// TwinCAT 3 PLC project Testing
// ProgramVersion: 3.1.4026.26
// libraries:
//   Tc2_Standard, 3.4.7.0 (Beckhoff Automation GmbH)
//   Tc2_System, 3.10.2.0 (Beckhoff Automation GmbH)
//   [TcForge], 2.0.0.0 (Home)
//   TcUnit, 1.3.0.0 (www.tcunit.org)
//   [TcForgeExample], 2.0.0.0 (Home)
// project tree:
//   Testing/POUs/ FB_ControlLoopFixture.TcPOU, FB_AnalogOutputRestart_Probe.TcPOU, FB_AlarmRestart_Probe.TcPOU, FB_RpcContext_Probe.TcPOU, FB_OutputRestart_Probe.TcPOU, MAIN.TcPOU, FB_DeviceBase_Probe.TcPOU, FB_StateMachine_Probe.TcPOU
//   Testing/Tests/ FB_RegulatoryControl_Edge_Test.TcPOU, FB_RegulatoryControl_Test.TcPOU, FB_HysteresisControl_Test.TcPOU, FB_ExecutionContinuity_Test.TcPOU, FB_DigitalInputLifecycle_Test.TcPOU, FB_AlarmValidity_Test.TcPOU, FB_FilterLifecycle_Test.TcPOU, FB_PolicyNumeric_Test.TcPOU, FB_OutputConfiguration_Test.TcPOU, FB_IOQualityMonitor_Test.TcPOU, FB_InputLifecycle_Test.TcPOU, FB_OperatorMailbox_Test.TcPOU, FB_CommandValidation_Test.TcPOU, FB_ReferenceMachine_Test.TcPOU, FB_SequenceIntegrity_Test.TcPOU, FB_Foundation_Test.TcPOU, FB_CyclicFoundation_Test.TcPOU, FB_F_ValidateRequester_Test.TcPOU, FB_BitMatrix64_Test.TcPOU, FB_Permissives_Test.TcPOU, FB_Interlock_Test.TcPOU, FB_AlarmSimple_Test.TcPOU, FB_AlarmLimit_Test.TcPOU, FB_DeviceBase_Test.TcPOU, FB_LPF_FirstOrder_IIR_Test.TcPOU, FB_DigitalOutput_Test.TcPOU, FB_DigitalInput_Test.TcPOU, FB_TwoPosActuator_Test.TcPOU, FB_AnalogInput_Test.TcPOU, FB_AnalogOutput_Test.TcPOU, FB_AlarmThreshold_Test.TcPOU, FB_AlarmDeviation_Test.TcPOU, FB_Step_Test.TcPOU, FB_StateMachine_Test.TcPOU, FB_AssemblyStation_Test.TcPOU
//   Testing/ Testing.TcTTO
// (motion and I/O tree: see PLC project tcforge)
// real-time tasks:
//   TASK Testing: cycle T#10ms, priority 2, ADS port 351
//   TASK PlcTask: cycle T#10ms, priority 1, ADS port 350

CONFIGURATION Testing
    RESOURCE PLC ON TwinCAT3
        TASK Testing(INTERVAL := T#10ms, PRIORITY := 2);
        PROGRAM MAIN WITH Testing : MAIN;
    END_RESOURCE
END_CONFIGURATION

// ---- Testing/POUs/MAIN.TcPOU
PROGRAM MAIN
VAR
    controlLoopFixture : FB_ControlLoopFixture;
    regulatoryControlEdge : FB_RegulatoryControl_Edge_Test;
    regulatoryControl : FB_RegulatoryControl_Test;
    hysteresisControl : FB_HysteresisControl_Test;
    executionContinuity : FB_ExecutionContinuity_Test;
    digitalInputLifecycle : FB_DigitalInputLifecycle_Test;
    alarmValidity : FB_AlarmValidity_Test;
    filterLifecycle : FB_FilterLifecycle_Test;
    policyNumeric : FB_PolicyNumeric_Test;
    outputConfiguration : FB_OutputConfiguration_Test;
    ioQuality : FB_IOQualityMonitor_Test;
    inputLifecycle : FB_InputLifecycle_Test;
    simulation : FB_SimulationBridge;
    operatorMailbox : FB_OperatorMailbox_Test;
    rpcOutput : TcForge.FB_DigitalOutput;
    rpcUninitialized : TcForge.FB_DigitalOutput;
    enableRpcPump : BOOL := TRUE;
    commandValidation : FB_CommandValidation_Test;
    rpcContext : FB_RpcContext_Probe;
    assemblyStation : FB_AssemblyStation_Test;
    referenceMachine : FB_ReferenceMachine_Test;
    sequenceIntegrity : FB_SequenceIntegrity_Test;
    foundation : FB_Foundation_Test;
    cyclicFoundation : FB_CyclicFoundation_Test;
    fbValidateRequester_Test : FB_F_ValidateRequester_Test;
    fbBitMatrix64_Test       : FB_BitMatrix64_Test;
    fbPermissives_Test       : FB_Permissives_Test;
    fbInterlock_Test         : FB_Interlock_Test;
    fbAlarmSimple_Test       : FB_AlarmSimple_Test;
    fbAlarmLimit_Test        : FB_AlarmLimit_Test;
    fbDeviceBase_Test        : FB_DeviceBase_Test;
    fbLpfFirstOrder_Test     : FB_LPF_FirstOrder_IIR_Test;
    fbDigitalOutput_Test     : FB_DigitalOutput_Test;
    fbDigitalInput_Test      : FB_DigitalInput_Test;
    fbTwoPosActuator_Test    : FB_TwoPosActuator_Test;
    fbAnalogInput_Test       : FB_AnalogInput_Test;
    fbAnalogOutput_Test      : FB_AnalogOutput_Test;
    fbAlarmThreshold_Test    : FB_AlarmThreshold_Test;
    fbAlarmDeviation_Test    : FB_AlarmDeviation_Test;
    fbStep_Test              : FB_Step_Test;
    fbStateMachine_Test      : FB_StateMachine_Test;
END_VAR

controlLoopFixture();
simulation();
rpcContext();
IF enableRpcPump THEN rpcOutput(); END_IF;
TcUnit.RUN();

END_PROGRAM

// ---- Testing/POUs/FB_ControlLoopFixture.TcPOU
// Bench-only ADS surface for a generic first-order analog plant. There is no
// physical IO binding or operator command path. The Python runner writes the
// payload first and requestFrame last; the cyclic owner copies one complete
// frame, computes PID, publishes the result, then acknowledges appliedFrame.
FUNCTION_BLOCK FB_ControlLoopFixture
VAR
    // Test-writer fields. One monotonically increasing frame is accepted at a time.
    requestFrame    : UDINT;
    requestEnable   : BOOL;
    requestPv       : REAL;
    requestQuality  : USINT;
    requestSetpoint : REAL;

    // Stable until the next accepted frame or the 500 ms feed watchdog expires.
    appliedFrame    : UDINT;
    rejectedFrame   : UDINT;
    outputCv        : REAL;
    ready           : BOOL;
    reason          : TcForge.E_ControlReason;
    watchdogExpired : BOOL;
    watchdogTrips   : UDINT;
    ownerTask       : DINT;
    cycleCounter    : UDINT;

    _pid            : TcForge.FB_PID_Full;
    _cfg            : TcForge.ST_PID_Full_Cfg;
    _watchdog       : TON;
    _wasExpired     : BOOL;
    _activeEnable   : BOOL;
    _activePv       : REAL;
    _activeQuality  : TcForge.E_IO_Quality := TcForge.E_IO_Quality.UNKNOWN;
    _activeSp       : REAL;
    _frameFault     : BOOL;
    accepted        : BOOL;
    expectedFrame   : UDINT;
    pendingFrame    : UDINT;
END_VAR

ownerTask := Tc2_System.GETCURTASKINDEXEX();
cycleCounter := cycleCounter + 1;
accepted := FALSE;

// The final frame write is the commit marker. Old or skipped frame numbers
// invalidate the feed instead of leaving the previous regulator demand live.
IF appliedFrame = UDINT#16#FFFFFFFF THEN
    expectedFrame := 0;
ELSE
    expectedFrame := appliedFrame + 1;
END_IF;

IF requestFrame <> appliedFrame THEN
    IF requestFrame = expectedFrame THEN
        _activeEnable := requestEnable;
        _activePv := requestPv;
        _activeSp := requestSetpoint;
        _activeQuality := TcForge.E_IO_Quality.BAD;
        IF requestQuality = 2 THEN
            _activeQuality := TcForge.E_IO_Quality.GOOD;
        END_IF;

        pendingFrame := requestFrame;
        _frameFault := FALSE;
        accepted := TRUE;
    ELSE
        rejectedFrame := requestFrame;
        _frameFault := TRUE;
    END_IF;
END_IF;

_watchdog(IN := NOT accepted, PT := T#500MS);
watchdogExpired := _watchdog.Q;
IF watchdogExpired AND NOT _wasExpired THEN
    watchdogTrips := watchdogTrips + 1;
END_IF;
_wasExpired := watchdogExpired;

// Fixed, bounded tuning makes the test process generic and reproducible.
// The task period is read from the owning PLC task, not from ADS pacing.
_cfg.kp := 2.0;
_cfg.ki := 1.0;
_cfg.kd := 0.0;
_cfg.cvMin := 0.0;
_cfg.cvMax := 100.0;
_cfg.safeCv := 0.0;
_cfg.cycleTime := T#0MS;
_cfg.maxDt := T#100MS;

_pid(
    enable := _activeEnable AND NOT watchdogExpired AND NOT _frameFault,
    pv := _activePv,
    pvQuality := _activeQuality,
    setpoint := _activeSp,
    cfg := _cfg
);
outputCv := _pid.outCv;
ready := _pid.sts.ready;
reason := _pid.sts.reason;

// Publish acknowledgement after the CV and status for this frame.
IF accepted THEN
    appliedFrame := pendingFrame;
END_IF;

END_FUNCTION_BLOCK

// ---- Testing/Tests/FB_RegulatoryControl_Edge_Test.TcPOU
// Exercises mode transitions and boundary cases beyond the basic control suite.
FUNCTION_BLOCK FB_RegulatoryControl_Edge_Test EXTENDS TcUnit.FB_TestSuite
VAR
    _done : BOOL;
END_VAR

IF _done THEN
    RETURN;
END_IF;

StandardFormUsesIntegralTime();
DerivativeFiltersPvWithoutSetpointKick();
LowerLimitUnwindsOnReversal();
HoldAndTrackReleaseWithoutStep();
InvalidConfigurationAndTimingFailSafe();
TemperatureManualDutyAndPeriodEdit();
TemperatureRejectsInvalidConfiguration();
SwitchingPvRecoversAfterQualityLoss();
SwitchingContractClearsOldStatus();

_done := TRUE;

METHOD PRIVATE StandardFormUsesIntegralTime
VAR
    fb : TcForge.FB_PID_Full;
END_VAR
TEST('StandardFormUsesIntegralTime');

fb.cfg.standardForm := TRUE;
fb.cfg.kp := 2.0;
fb.cfg.integralTime := T#1S;
fb.cfg.cycleTime := T#100MS;
fb(enable := TRUE, pv := 0.0, pvQuality := TcForge.E_IO_Quality.GOOD, setpoint := 10.0);

AssertEquals_REAL(22.0, fb.outCv, 0.02, 'Standard form uses Kp/Ti for integral gain');
fb();
AssertEquals_REAL(24.0, fb.outCv, 0.02, 'Integral time advances the CV each cycle');

TEST_FINISHED();
END_METHOD

METHOD PRIVATE DerivativeFiltersPvWithoutSetpointKick
VAR
    fb : TcForge.FB_PID_Full;
END_VAR
TEST('DerivativeFiltersPvWithoutSetpointKick');

fb.cfg.kp := 0.0;
fb.cfg.kd := 1.0;
fb.cfg.derivativeTau := T#100MS;
fb.cfg.cvMin := -100.0;
fb.cfg.cycleTime := T#100MS;
fb(enable := TRUE, pv := 0.0, pvQuality := TcForge.E_IO_Quality.GOOD, setpoint := 0.0);

fb(pv := 1.0);
AssertEquals_REAL(-5.0, fb.outCv, 0.1, 'First-order filter halves the PV derivative');

fb(setpoint := 50.0);
AssertEquals_REAL(-2.5, fb.outCv, 0.1, 'Setpoint step does not enter PV derivative');

TEST_FINISHED();
END_METHOD

METHOD PRIVATE LowerLimitUnwindsOnReversal
VAR
    fb : TcForge.FB_PID_Full;
END_VAR
TEST('LowerLimitUnwindsOnReversal');

fb.cfg.kp := 0.0;
fb.cfg.ki := 1.0;
fb.cfg.cvMin := -2.0;
fb.cfg.cvMax := 2.0;
fb.cfg.cycleTime := T#100MS;
fb(enable := TRUE, pv := 0.0, pvQuality := TcForge.E_IO_Quality.GOOD, setpoint := -10.0);

fb();
fb();
AssertTrue(fb.sts.saturated, 'Further negative integration reports saturation');
AssertEquals_REAL(-2.0, fb.outCv, 0.02, 'Lower CV boundary is reached without windup');

fb(setpoint := 10.0);
AssertEquals_REAL(-1.0, fb.outCv, 0.02, 'Error reversal immediately unwinds integral');

TEST_FINISHED();
END_METHOD

METHOD PRIVATE HoldAndTrackReleaseWithoutStep
VAR
    fb : TcForge.FB_PID_Full;
END_VAR
TEST('HoldAndTrackReleaseWithoutStep');

fb.cfg.cycleTime := T#100MS;
fb(enable := TRUE, pv := 0.0, pvQuality := TcForge.E_IO_Quality.GOOD, setpoint := 20.0);
AssertEquals_REAL(20.0, fb.outCv, 0.01, 'Precondition: automatic CV');

fb(hold := TRUE, setpoint := 40.0);
AssertEquals_REAL(20.0, fb.outCv, 0.01, 'Hold keeps the last CV');
AssertTrue(fb.sts.reason = TcForge.E_ControlReason.Held, 'Hold mode is visible');

fb(track := TRUE, trackCv := 35.0);
AssertEquals_REAL(35.0, fb.outCv, 0.01, 'One-scan tracking takes the requested CV');

fb(track := FALSE, hold := FALSE);
AssertEquals_REAL(35.0, fb.outCv, 0.01, 'Automatic release uses tracked integral bias');

TEST_FINISHED();
END_METHOD

METHOD PRIVATE InvalidConfigurationAndTimingFailSafe
VAR
    fb : TcForge.FB_PID_Full;
END_VAR
TEST('InvalidConfigurationAndTimingFailSafe');

fb.cfg.cvMin := 100.0;
fb.cfg.cvMax := 0.0;
fb(enable := TRUE, pv := 0.0, pvQuality := TcForge.E_IO_Quality.GOOD, setpoint := 20.0);
AssertFalse(fb.sts.ready, 'Reversed CV limits cannot run');
AssertTrue(fb.sts.reason = TcForge.E_ControlReason.InvalidConfig, 'Invalid limits are diagnosed');
AssertEquals_REAL(0.0, fb.outCv, 0.001, 'Invalid configuration returns zero');

fb.cfg.cvMin := 0.0;
fb.cfg.cvMax := 100.0;
fb.cfg.cycleTime := T#2S;
fb();
AssertTrue(fb.sts.reason = TcForge.E_ControlReason.InvalidTiming, 'Oversize declared task interval is rejected');

fb.cfg.cycleTime := T#100MS;
fb();
AssertTrue(fb.sts.ready, 'Corrected timing starts a fresh controller');

fb(pvQuality := TcForge.E_IO_Quality.BAD);
AssertEquals_REAL(0.0, fb.outCv, 0.001, 'Bad quality immediately returns safe CV');

TEST_FINISHED();
END_METHOD

METHOD PRIVATE TemperatureManualDutyAndPeriodEdit
VAR
    fb : TcForge.FB_TempController;
    index : INT;
END_VAR
TEST('TemperatureManualDutyAndPeriodEdit');

fb.cfg.pid.cycleTime := T#100MS;
fb.cfg.pwmPeriod := T#1S;
fb(enable := TRUE, pv := 0.0, pvQuality := TcForge.E_IO_Quality.GOOD,
    setpoint := 25.0, manual := TRUE, manualDuty := 60.0);
AssertEquals_REAL(60.0, fb.outDuty, 0.01, 'Manual duty is applied as percent');

FOR index := 1 TO 7 DO
    fb();
END_FOR;
AssertFalse(fb.outOn, 'PWM reaches its OFF interval');

fb.cfg.pwmPeriod := T#2S;
fb();
AssertTrue(fb.outOn, 'Period edit restarts a bounded PWM window');

fb.cfg.pwmPeriod := T#50MS;
fb();
AssertFalse(fb.sts.ready, 'Too-short period is rejected');
AssertFalse(fb.outOn, 'Invalid period de-energizes PWM');

fb.cfg.pwmPeriod := T#1S;
fb();
AssertTrue(fb.sts.ready AND fb.outOn, 'Recovery starts a fresh ON window');

TEST_FINISHED();
END_METHOD

METHOD PRIVATE TemperatureRejectsInvalidConfiguration
VAR
    fb : TcForge.FB_TempController;
    invalid : REAL;
    bits : DWORD := DWORD#16#7F800001; // Signaling NaN; classify bits before comparison.
END_VAR
TEST('TemperatureRejectsInvalidConfiguration');

fb.cfg.pid.cvMin := -1.0;
fb.cfg.pid.cycleTime := T#100MS;
fb(enable := TRUE, pv := 0.0, pvQuality := TcForge.E_IO_Quality.GOOD, setpoint := 80.0);
AssertFalse(fb.sts.ready OR fb.outOn, 'Non-percent CV contract fails OFF');

fb.cfg.pid.cvMin := 0.0;
fb();
AssertTrue(fb.sts.ready AND fb.outOn, 'Valid percent contract can recover');

Tc2_System.MEMCPY(destAddr := ADR(invalid), srcAddr := ADR(bits), n := SIZEOF(invalid));
fb.cfg.standbySetpoint := invalid;
fb();
AssertFalse(fb.sts.ready OR fb.outOn, 'Nonfinite standby SP fails OFF even before use');

fb.cfg.standbySetpoint := 25.0;
fb();
AssertTrue(fb.sts.ready, 'Finite standby SP can recover');

TEST_FINISHED();
END_METHOD

METHOD PRIVATE SwitchingPvRecoversAfterQualityLoss
VAR
    fb : TcForge.FB_SwitchingPvPid;
END_VAR
TEST('SwitchingPvRecoversAfterQualityLoss');

fb.cfg.pv1.cycleTime := T#100MS;
fb.cfg.pv2.cycleTime := T#100MS;
fb(enable := TRUE, source := TcForge.E_PvSource.PV1,
    pv1 := 0.0, quality1 := TcForge.E_IO_Quality.GOOD, setpoint1 := 30.0,
    pv2 := 0.0, quality2 := TcForge.E_IO_Quality.BAD, setpoint2 := 40.0);
AssertEquals_REAL(30.0, fb.outCv, 0.01, 'PV1 is initially authoritative');

fb(source := TcForge.E_PvSource.PV2);
AssertFalse(fb.sts.ready, 'Selected bad PV cannot retain previous output');
AssertEquals_REAL(0.0, fb.outCv, 0.01, 'Bad selected PV returns common safe CV');

fb(quality2 := TcForge.E_IO_Quality.GOOD);
AssertEquals_REAL(40.0, fb.outCv, 0.01, 'Recovery uses fresh PV2 tuning, not stale CV');

TEST_FINISHED();
END_METHOD

METHOD PRIVATE SwitchingContractClearsOldStatus
VAR
    fb : TcForge.FB_SwitchingPvPid;
END_VAR
TEST('SwitchingContractClearsOldStatus');

fb.cfg.pv1.cycleTime := T#100MS;
fb.cfg.pv2.cycleTime := T#100MS;
fb(enable := TRUE, pv1 := 0.0, quality1 := TcForge.E_IO_Quality.GOOD, setpoint1 := 20.0);
AssertTrue(fb.sts.pid.ready, 'Precondition: PID status ready');

fb.cfg.pv2.cvMax := 80.0;
fb();
AssertFalse(fb.sts.ready OR fb.sts.pid.ready, 'Invalid shared contract clears old ready status');
AssertEquals_REAL(0.0, fb.outCv, 0.01, 'Invalid contract fails OFF');

fb.cfg.pv2.cvMax := 100.0;
fb();
AssertTrue(fb.sts.ready, 'Restored output contract can recover');

TEST_FINISHED();
END_METHOD

END_FUNCTION_BLOCK

// ---- Testing/Tests/FB_RegulatoryControl_Test.TcPOU
FUNCTION_BLOCK FB_RegulatoryControl_Test EXTENDS TcUnit.FB_TestSuite
VAR
    _done : BOOL;
END_VAR

IF _done THEN RETURN; END_IF;

BangBangMapsDemand();
PidProportionalAndReverse();
PidIntegralAndAntiWindup();
PidQualityAndManual();
PidSetpointAndCvRamps();
PidExceptionalInputFailsSafe();
TemperaturePwmAndStandby();
TemperatureQualityFailsOff();
SwitchingTracksCv();
SwitchingRejectsIncompatibleOutput();

_done := TRUE;

METHOD PRIVATE BangBangMapsDemand
VAR fb : TcForge.FB_BangBang; END_VAR
TEST('BangBangMapsDemand');
fb.cfg.hysteresis.low := 10.0;
fb.cfg.hysteresis.high := 20.0;
fb.cfg.lowValue := 5.0;
fb.cfg.highValue := 75.0;

fb(enable := TRUE, pv := 5.0, pvQuality := TcForge.E_IO_Quality.GOOD);
AssertTrue(fb.outDemand, 'Low PV requests the high mapped value');
AssertEquals_REAL(75.0, fb.outCv, 0.001, 'High value maps demand ON');

fb(pv := 20.0);
AssertFalse(fb.outDemand, 'High threshold clears demand');
AssertEquals_REAL(5.0, fb.outCv, 0.001, 'Low value maps demand OFF');

fb(pvQuality := TcForge.E_IO_Quality.BAD);
AssertFalse(fb.sts.ready, 'Bad quality invalidates mapped CV');
AssertEquals_REAL(0.0, fb.outCv, 0.001, 'Unusable mapping fails to zero');
TEST_FINISHED();
END_METHOD

METHOD PRIVATE PidProportionalAndReverse
VAR fb : TcForge.FB_PID_Full; END_VAR
TEST('PidProportionalAndReverse');
fb.cfg.kp := 2.0;
fb.cfg.cycleTime := T#100MS;
fb(enable := TRUE, pv := 20.0, pvQuality := TcForge.E_IO_Quality.GOOD, setpoint := 30.0);
AssertTrue(fb.sts.ready, 'Finite configured PID is ready');
AssertEquals_REAL(20.0, fb.outCv, 0.001, 'Direct P term drives CV');

fb.cfg.reverseActing := TRUE;
fb(pv := 30.0, setpoint := 20.0);
AssertFalse(fb.sts.ready, 'Tuning direction edit gets a safe scan');
fb();
AssertEquals_REAL(20.0, fb.outCv, 0.001, 'Reverse action changes error sign');
TEST_FINISHED();
END_METHOD

METHOD PRIVATE PidIntegralAndAntiWindup
VAR fb : TcForge.FB_PID_Full; END_VAR
TEST('PidIntegralAndAntiWindup');
fb.cfg.kp := 0.0;
fb.cfg.ki := 1.0;
fb.cfg.cycleTime := T#100MS;
fb(enable := TRUE, pv := 0.0, pvQuality := TcForge.E_IO_Quality.GOOD, setpoint := 10.0);
AssertEquals_REAL(1.0, fb.outCv, 0.001, 'Integral accumulates error times seconds');

fb();
AssertEquals_REAL(2.0, fb.outCv, 0.001, 'Integral advances by one output unit per scan');

fb.cfg.cvMax := 2.0;
fb();
AssertFalse(fb.sts.ready, 'CV limit edit invalidates old integral history');
fb();
AssertEquals_REAL(1.0, fb.outCv, 0.001, 'Reset history resumes from a fresh integral');
fb();
fb();
AssertTrue(fb.sts.saturated, 'Further integration is blocked at the CV limit');
AssertEquals_REAL(2.0, fb.outCv, 0.001, 'CV stays within the edited limit');
TEST_FINISHED();
END_METHOD

METHOD PRIVATE PidQualityAndManual
VAR fb : TcForge.FB_PID_Full; END_VAR
TEST('PidQualityAndManual');
fb.cfg.kp := 1.0;
fb.cfg.ki := 1.0;
fb.cfg.cycleTime := T#100MS;
fb(enable := TRUE, pv := 0.0, pvQuality := TcForge.E_IO_Quality.GOOD, setpoint := 10.0);
AssertTrue(fb.outCv > 0.0, 'Precondition: automatic CV is positive');

fb(manual := TRUE, manualCv := 40.0);
AssertEquals_REAL(40.0, fb.outCv, 0.001, 'Manual request is limited and published');
AssertTrue(fb.sts.reason = TcForge.E_ControlReason.Manual, 'Manual mode is visible');

fb(manual := FALSE);
AssertTrue(fb.outCv >= 40.0 AND fb.outCv < 42.0, 'Automatic resumes near tracked manual CV');

fb(pvQuality := TcForge.E_IO_Quality.BAD);
AssertEquals_REAL(0.0, fb.outCv, 0.001, 'Bad measurement immediately returns safe CV');
AssertFalse(fb.sts.ready, 'Bad quality cannot report ready');
TEST_FINISHED();
END_METHOD

METHOD PRIVATE PidSetpointAndCvRamps
VAR fb : TcForge.FB_PID_Full; END_VAR
TEST('PidSetpointAndCvRamps');
fb.cfg.kp := 1.0;
fb.cfg.spRateUp := 10.0;
fb.cfg.cvRateUp := 5.0;
fb.cfg.cycleTime := T#100MS;
fb(enable := TRUE, pv := 0.0, pvQuality := TcForge.E_IO_Quality.GOOD, setpoint := 0.0);

fb(setpoint := 10.0);
AssertEquals_REAL(1.0, fb.sts.spApplied, 0.001, 'SP ramp uses engineering units per second');
AssertEquals_REAL(0.5, fb.outCv, 0.001, 'CV ramp uses output units per second');
AssertTrue(fb.sts.spRamping AND fb.sts.cvRamping, 'Both active ramps are reported');
TEST_FINISHED();
END_METHOD

METHOD PRIVATE PidExceptionalInputFailsSafe
VAR
    fb : TcForge.FB_PID_Full;
    invalid : REAL;
    bits : DWORD := DWORD#16#7F800001; // Signaling NaN.
END_VAR
TEST('PidExceptionalInputFailsSafe');
fb.cfg.cycleTime := T#100MS;
fb(enable := TRUE, pv := 0.0, pvQuality := TcForge.E_IO_Quality.GOOD, setpoint := 20.0);
AssertTrue(fb.sts.ready, 'Precondition: valid PID');

Tc2_System.MEMCPY(destAddr := ADR(invalid), srcAddr := ADR(bits), n := SIZEOF(invalid));
fb(pv := invalid);
AssertFalse(fb.sts.ready, 'Signaling NaN is rejected before arithmetic');
AssertEquals_REAL(0.0, fb.outCv, 0.001, 'Rejected PV fails to safe CV');

fb(pv := 0.0);
AssertTrue(fb.sts.ready, 'Fresh finite PV can recover');
TEST_FINISHED();
END_METHOD

METHOD PRIVATE TemperaturePwmAndStandby
VAR fb : TcForge.FB_TempController; i : INT; END_VAR
TEST('TemperaturePwmAndStandby');
fb.cfg.pid.kp := 1.0;
fb.cfg.pid.cycleTime := T#100MS;
fb.cfg.pwmPeriod := T#1S;
fb.cfg.standbyEnabled := TRUE;
fb.cfg.standbySetpoint := 0.0;
fb(enable := TRUE, pv := 0.0, pvQuality := TcForge.E_IO_Quality.GOOD, setpoint := 50.0);
AssertEquals_REAL(50.0, fb.outDuty, 0.001, 'PID CV maps to 50 percent duty');
AssertTrue(fb.outOn, 'First half of PWM window is ON');

FOR i := 1 TO 5 DO fb(); END_FOR;
AssertFalse(fb.outOn, 'Second half of PWM window is OFF');

fb(standby := TRUE);
AssertTrue(fb.sts.standbyActive, 'Standby selects its own setpoint');
AssertEquals_REAL(0.0, fb.outDuty, 0.001, 'Standby zero setpoint removes heating demand');
AssertFalse(fb.outOn, 'Zero duty is OFF');
TEST_FINISHED();
END_METHOD

METHOD PRIVATE TemperatureQualityFailsOff
VAR fb : TcForge.FB_TempController; END_VAR
TEST('TemperatureQualityFailsOff');
fb.cfg.pid.cycleTime := T#100MS;
fb(enable := TRUE, pv := 0.0, pvQuality := TcForge.E_IO_Quality.GOOD, setpoint := 100.0);
AssertTrue(fb.outOn, 'Precondition: full-duty output ON');

fb(pvQuality := TcForge.E_IO_Quality.BAD);
AssertFalse(fb.outOn, 'Sensor loss removes PWM in the same scan');
AssertEquals_REAL(0.0, fb.outDuty, 0.001, 'Sensor loss returns zero duty');
AssertFalse(fb.sts.ready, 'Sensor loss cannot report ready');
TEST_FINISHED();
END_METHOD

METHOD PRIVATE SwitchingTracksCv
VAR fb : TcForge.FB_SwitchingPvPid; END_VAR
TEST('SwitchingTracksCv');
fb.cfg.pv1.cycleTime := T#100MS;
fb.cfg.pv2.cycleTime := T#100MS;
fb.cfg.pv2.ki := 1.0;
fb(enable := TRUE,
   source := TcForge.E_PvSource.PV1,
   pv1 := 0.0, quality1 := TcForge.E_IO_Quality.GOOD, setpoint1 := 20.0,
   pv2 := 0.0, quality2 := TcForge.E_IO_Quality.GOOD, setpoint2 := 40.0);
AssertEquals_REAL(20.0, fb.outCv, 0.001, 'PV1 regulates the shared output');

fb(source := TcForge.E_PvSource.PV2);
AssertTrue(fb.sts.sourceChanged, 'Selection change is published');
AssertEquals_REAL(20.0, fb.outCv, 0.001, 'PV2 tracks the previous CV for one scan');

fb();
AssertTrue(fb.outCv > 20.0 AND fb.outCv < 25.0, 'Selected PID resumes regulation');

fb(quality2 := TcForge.E_IO_Quality.BAD);
AssertFalse(fb.sts.ready, 'Selected bad PV invalidates the output');
AssertEquals_REAL(0.0, fb.outCv, 0.001, 'Selected bad PV uses the common safe CV');
TEST_FINISHED();
END_METHOD

METHOD PRIVATE SwitchingRejectsIncompatibleOutput
VAR fb : TcForge.FB_SwitchingPvPid; END_VAR
TEST('SwitchingRejectsIncompatibleOutput');
fb.cfg.pv1.cycleTime := T#100MS;
fb.cfg.pv2.cycleTime := T#100MS;
fb.cfg.pv2.cvMax := 80.0;
fb(enable := TRUE, pv1 := 0.0,
   quality1 := TcForge.E_IO_Quality.GOOD, setpoint1 := 50.0);
AssertFalse(fb.sts.ready, 'Different CV ranges cannot drive the same output');
AssertEquals_REAL(0.0, fb.outCv, 0.001, 'Mismatched output contract fails OFF');
TEST_FINISHED();
END_METHOD

END_FUNCTION_BLOCK

// ---- Testing/Tests/FB_HysteresisControl_Test.TcPOU
FUNCTION_BLOCK FB_HysteresisControl_Test EXTENDS TcUnit.FB_TestSuite
VAR
    _done : BOOL;
END_VAR

IF _done THEN
    RETURN;
END_IF;

DefaultRequiresConfiguration();
LowActingDeadband();
HighActingDeadband();
QualityLossClearsDemand();
ConfigChangeClearsDemand();
ExceptionalValuesFailOff();
DisableClearsDemand();

_done := TRUE;

METHOD PRIVATE DefaultRequiresConfiguration
VAR
    fb : TcForge.FB_HysteresisControl;
END_VAR
TEST('DefaultRequiresConfiguration');

fb(enable := TRUE, pv := 15.0, pvQuality := TcForge.E_IO_Quality.GOOD);
AssertFalse(fb.outDemand, 'Equal default thresholds cannot energize');
AssertTrue(fb.sts.reason = TcForge.E_HysteresisReason.InvalidConfig, 'Invalid defaults are visible');

fb.cfg.low := 10.0;
fb.cfg.high := 20.0;
fb();
AssertTrue(fb.sts.ready, 'Configured finite PV is ready');
AssertFalse(fb.outDemand, 'Startup inside the deadband starts OFF');

TEST_FINISHED();
END_METHOD

METHOD PRIVATE LowActingDeadband
VAR
    fb : TcForge.FB_HysteresisControl;
END_VAR
TEST('LowActingDeadband');

fb.cfg.low := 10.0;
fb.cfg.high := 20.0;
fb(enable := TRUE, pv := 5.0, pvQuality := TcForge.E_IO_Quality.GOOD);
AssertTrue(fb.outDemand, 'Heating demand turns ON below low threshold');

fb(pv := 15.0);
AssertTrue(fb.outDemand AND fb.sts.inDeadband, 'Demand holds ON inside deadband');

fb(pv := 20.0);
AssertFalse(fb.outDemand, 'Demand turns OFF at high threshold');

fb(pv := 15.0);
AssertFalse(fb.outDemand, 'Deadband also retains OFF state');

fb(pv := 10.0);
AssertTrue(fb.outDemand, 'Demand turns ON at low threshold');

TEST_FINISHED();
END_METHOD

METHOD PRIVATE HighActingDeadband
VAR
    fb : TcForge.FB_HysteresisControl;
END_VAR
TEST('HighActingDeadband');

fb.cfg.low := 10.0;
fb.cfg.high := 20.0;
fb.cfg.onBelowLow := FALSE;
fb(enable := TRUE, pv := 25.0, pvQuality := TcForge.E_IO_Quality.GOOD);
AssertTrue(fb.outDemand, 'Cooling demand turns ON above high threshold');

fb(pv := 15.0);
AssertTrue(fb.outDemand, 'Cooling demand holds ON inside deadband');

fb(pv := 10.0);
AssertFalse(fb.outDemand, 'Cooling demand turns OFF at low threshold');

fb(pv := 15.0);
AssertFalse(fb.outDemand, 'Cooling deadband retains OFF state');

TEST_FINISHED();
END_METHOD

METHOD PRIVATE QualityLossClearsDemand
VAR
    fb : TcForge.FB_HysteresisControl;
END_VAR
TEST('QualityLossClearsDemand');

fb.cfg.low := 10.0;
fb.cfg.high := 20.0;
fb(enable := TRUE, pv := 5.0, pvQuality := TcForge.E_IO_Quality.GOOD);
AssertTrue(fb.outDemand, 'Precondition: demand ON');

fb(pvQuality := TcForge.E_IO_Quality.BAD);
AssertFalse(fb.outDemand, 'Quality loss removes demand in the same scan');
AssertTrue(fb.sts.reason = TcForge.E_HysteresisReason.BadQuality, 'Quality loss is diagnosed');

fb(pv := 15.0, pvQuality := TcForge.E_IO_Quality.GOOD);
AssertFalse(fb.outDemand, 'Recovery inside deadband cannot restore stale ON intent');

fb(pv := 10.0);
AssertTrue(fb.outDemand, 'Fresh threshold crossing may demand ON');

TEST_FINISHED();
END_METHOD

METHOD PRIVATE ConfigChangeClearsDemand
VAR
    fb : TcForge.FB_HysteresisControl;
END_VAR
TEST('ConfigChangeClearsDemand');

fb.cfg.low := 10.0;
fb.cfg.high := 20.0;
fb(enable := TRUE, pv := 5.0, pvQuality := TcForge.E_IO_Quality.GOOD);
AssertTrue(fb.outDemand, 'Precondition: old recipe demands ON');

fb.cfg.low := 0.0;
fb(pv := 5.0);
AssertFalse(fb.outDemand, 'Changed threshold cannot inherit old ON state in deadband');

fb.cfg.onBelowLow := FALSE;
fb();
AssertFalse(fb.outDemand, 'Changed direction also starts from OFF');

fb(pv := 20.0);
AssertTrue(fb.outDemand, 'New direction can turn ON at its threshold');

TEST_FINISHED();
END_METHOD

METHOD PRIVATE ExceptionalValuesFailOff
VAR
    fb : TcForge.FB_HysteresisControl;
    invalid : REAL;
    bits : DWORD := DWORD#16#7F800001; // Signaling NaN; never compare as REAL.
END_VAR
TEST('ExceptionalValuesFailOff');

fb.cfg.low := 10.0;
fb.cfg.high := 20.0;
fb(enable := TRUE, pv := 5.0, pvQuality := TcForge.E_IO_Quality.GOOD);
AssertTrue(fb.outDemand, 'Precondition: demand ON');

Tc2_System.MEMCPY(destAddr := ADR(invalid), srcAddr := ADR(bits), n := SIZEOF(invalid));
fb(pv := invalid);
AssertFalse(fb.outDemand, 'Nonfinite PV fails OFF without a floating-point comparison');
AssertTrue(fb.sts.reason = TcForge.E_HysteresisReason.InvalidValue, 'Nonfinite PV is diagnosed');

fb(pv := 5.0);
AssertTrue(fb.outDemand, 'Fresh valid PV at threshold may restore demand');

fb.cfg.low := invalid;
fb();
AssertFalse(fb.outDemand, 'Nonfinite threshold fails OFF');
AssertTrue(fb.sts.reason = TcForge.E_HysteresisReason.InvalidConfig, 'Bad threshold is diagnosed');

TEST_FINISHED();
END_METHOD

METHOD PRIVATE DisableClearsDemand
VAR
    fb : TcForge.FB_HysteresisControl;
END_VAR
TEST('DisableClearsDemand');

fb.cfg.low := 10.0;
fb.cfg.high := 20.0;
fb(enable := TRUE, pv := 5.0, pvQuality := TcForge.E_IO_Quality.GOOD);
AssertTrue(fb.outDemand, 'Precondition: demand ON');

fb(enable := FALSE);
AssertFalse(fb.outDemand, 'Disable removes demand');
AssertTrue(fb.sts.reason = TcForge.E_HysteresisReason.Disabled, 'Disabled status is explicit');

fb(enable := TRUE, pv := 15.0);
AssertFalse(fb.outDemand, 'Re-enable inside deadband remains OFF');

TEST_FINISHED();
END_METHOD

END_FUNCTION_BLOCK

// ---- Testing/Tests/FB_ExecutionContinuity_Test.TcPOU
FUNCTION_BLOCK FB_ExecutionContinuity_Test EXTENDS TcUnit.FB_TestSuite
VAR done : BOOL; END_VAR

IF NOT done THEN
InitialObservationEstablishesBaseline();
ContinuousAndRepeatedCycle();
SkippedScanRequiresRecovery();
OnlineChangeDetectedWithoutGap();
TaskChangeAndInvalidContext();
CounterWrapAndReset();
CompatibleChangePreservesExecution();
CompatibleChangeCannotMaskGap();
CompatiblePolicyCannotMaskOwnerFailure();
done := TRUE; END_IF;

METHOD InitialObservationEstablishesBaseline
VAR fb : TcForge.FB_ExecutionContinuity; END_VAR
TEST('InitialObservationEstablishesBaseline');
fb(taskIndex := 1, cycleCounter := 99, onlineChangeCounter := 3); AssertFalse(Condition := fb.interrupted, Message := 'First sample establishes baseline');
TEST_FINISHED();
END_METHOD

METHOD ContinuousAndRepeatedCycle
VAR fb : TcForge.FB_ExecutionContinuity; END_VAR
TEST('ContinuousAndRepeatedCycle');
fb(taskIndex := 1, cycleCounter := 99); fb(cycleCounter := 100); AssertFalse(Condition := fb.interrupted, Message := 'Next scan continues'); fb(); AssertFalse(Condition := fb.interrupted, Message := 'Same scan observation is idempotent');
TEST_FINISHED();
END_METHOD

METHOD SkippedScanRequiresRecovery
VAR fb : TcForge.FB_ExecutionContinuity; END_VAR
TEST('SkippedScanRequiresRecovery');
fb(taskIndex := 1, cycleCounter := 99); fb(cycleCounter := 101); AssertTrue(Condition := fb.interrupted, Message := 'Missed execution detected'); fb(cycleCounter := 102); AssertFalse(Condition := fb.interrupted, Message := 'Caller must latch recovery; event is one scan');
TEST_FINISHED();
END_METHOD

METHOD OnlineChangeDetectedWithoutGap
VAR fb : TcForge.FB_ExecutionContinuity; END_VAR
TEST('OnlineChangeDetectedWithoutGap');
fb(taskIndex := 1, cycleCounter := 99, onlineChangeCounter := 3); fb(cycleCounter := 100, onlineChangeCounter := 4); AssertTrue(Condition := fb.interrupted, Message := 'Implementation-only online change detected');
TEST_FINISHED();
END_METHOD

METHOD TaskChangeAndInvalidContext
VAR fb : TcForge.FB_ExecutionContinuity; END_VAR
TEST('TaskChangeAndInvalidContext');
fb(taskIndex := 1, cycleCounter := 99); fb(taskIndex := 2, cycleCounter := 100); AssertTrue(Condition := fb.interrupted, Message := 'Different owner detected'); fb(taskIndex := 0); AssertTrue(Condition := fb.interrupted, Message := 'RPC or invalid context rejected');
TEST_FINISHED();
END_METHOD

METHOD CounterWrapAndReset
VAR fb : TcForge.FB_ExecutionContinuity; END_VAR
TEST('CounterWrapAndReset');
fb(taskIndex := 1, cycleCounter := UDINT#16#FFFFFFFF); fb(cycleCounter := 0); AssertFalse(Condition := fb.interrupted, Message := 'Natural wrap is continuous'); fb(cycleCounter := 99); fb(cycleCounter := 0); AssertTrue(Condition := fb.interrupted, Message := 'Counter discontinuity detected');
TEST_FINISHED();
END_METHOD

METHOD CompatibleChangePreservesExecution
VAR fb : TcForge.FB_ExecutionContinuity; END_VAR
TEST('CompatibleChangePreservesExecution');
fb(taskIndex := 1, cycleCounter := 99, onlineChangeCounter := 3, recoverOnOnlineChange := FALSE);
fb(cycleCounter := 100, onlineChangeCounter := 4);
AssertTrue(Condition := fb.onlineChanged, Message := 'Change remains observable');
AssertFalse(Condition := fb.executionInterrupted, Message := 'Online edit is not an execution gap');
AssertFalse(Condition := fb.interrupted, Message := 'Explicit compatible-edit policy preserves execution');
fb(cycleCounter := 101);
AssertFalse(Condition := fb.onlineChanged, Message := 'Change notification is a pulse');
TEST_FINISHED();
END_METHOD

METHOD CompatibleChangeCannotMaskGap
VAR fb : TcForge.FB_ExecutionContinuity; END_VAR
TEST('CompatibleChangeCannotMaskGap');
fb(taskIndex := 1, cycleCounter := 99, onlineChangeCounter := 3, recoverOnOnlineChange := FALSE);
fb(cycleCounter := 101, onlineChangeCounter := 4);
AssertTrue(Condition := fb.onlineChanged, Message := 'Simultaneous online edit observed');
AssertTrue(Condition := fb.executionInterrupted, Message := 'Gap remains a gap during online edit');
AssertTrue(Condition := fb.interrupted, Message := 'Compatible-edit policy cannot suppress recovery');
TEST_FINISHED();
END_METHOD

METHOD CompatiblePolicyCannotMaskOwnerFailure
VAR fb : TcForge.FB_ExecutionContinuity; END_VAR
TEST('CompatiblePolicyCannotMaskOwnerFailure');
fb(taskIndex := 1, cycleCounter := 99, recoverOnOnlineChange := FALSE);
fb(taskIndex := 2, cycleCounter := 100);
AssertTrue(Condition := fb.interrupted, Message := 'Owner conflict still requires recovery');
fb(taskIndex := 0);
AssertTrue(Condition := fb.executionInterrupted, Message := 'Invalid context still fails closed');
TEST_FINISHED();
END_METHOD

END_FUNCTION_BLOCK

// ---- Testing/Tests/FB_DigitalInputLifecycle_Test.TcPOU
FUNCTION_BLOCK FB_DigitalInputLifecycle_Test EXTENDS TcUnit.FB_TestSuite
VAR
BadQualityCannotCompleteRising_fb : TcForge.FB_DigitalInput;
BadQualityCannotCompleteRising_clock : TON;
BadQualityCannotCompleteRising_phase : UINT;
BadQualityCannotCompleteRising_done : BOOL;
BadQualityCannotCompleteFalling_fb : TcForge.FB_DigitalInput;
BadQualityCannotCompleteFalling_clock : TON;
BadQualityCannotCompleteFalling_phase : UINT;
BadQualityCannotCompleteFalling_done : BOOL;
ConfigChangeDiscardsDebounceCredit_fb : TcForge.FB_DigitalInput;
ConfigChangeDiscardsDebounceCredit_clock : TON;
ConfigChangeDiscardsDebounceCredit_phase : UINT;
ConfigChangeDiscardsDebounceCredit_done : BOOL;
_instantDone : BOOL;
END_VAR


BadQualityCannotCompleteRising();
BadQualityCannotCompleteFalling();
ConfigChangeDiscardsDebounceCredit();
IF NOT _instantDone THEN ReassignmentAndInvalidConfigHold(); _instantDone := TRUE; END_IF;

METHOD BadQualityCannotCompleteRising
IF BadQualityCannotCompleteRising_done THEN RETURN; END_IF;
TEST('BadQualityCannotCompleteRising');
CASE BadQualityCannotCompleteRising_phase OF
0:
    BadQualityCannotCompleteRising_fb(inSignal := FALSE);
    BadQualityCannotCompleteRising_fb.cfg.debounceOn := T#80MS; BadQualityCannotCompleteRising_fb.cfg.debounceOff := T#80MS;
    BadQualityCannotCompleteRising_fb(inSignal := TRUE);
    BadQualityCannotCompleteRising_fb(inpQuality := TcForge.E_IO_Quality.BAD);
    BadQualityCannotCompleteRising_phase := 1;
1:
    BadQualityCannotCompleteRising_clock(IN := TRUE, PT := T#150MS); BadQualityCannotCompleteRising_fb();
    IF BadQualityCannotCompleteRising_clock.Q THEN
        AssertEquals_BOOL(Expected := FALSE, Actual := BadQualityCannotCompleteRising_fb.sts.value, Message := 'Invalid elapsed time must hold established state');
        AssertFalse(Condition := BadQualityCannotCompleteRising_fb.sts.risingEdge OR BadQualityCannotCompleteRising_fb.sts.fallingEdge, Message := 'Invalid sample cannot emit edges');
        BadQualityCannotCompleteRising_clock(IN := FALSE); BadQualityCannotCompleteRising_fb(inpQuality := TcForge.E_IO_Quality.GOOD);
        AssertEquals_BOOL(Expected := FALSE, Actual := BadQualityCannotCompleteRising_fb.sts.value, Message := 'Recovery starts a full fresh transition delay');
        BadQualityCannotCompleteRising_phase := 2;
    END_IF;
2:
    BadQualityCannotCompleteRising_clock(IN := TRUE, PT := T#30MS); BadQualityCannotCompleteRising_fb();
    IF BadQualityCannotCompleteRising_clock.Q THEN
        AssertEquals_BOOL(Expected := FALSE, Actual := BadQualityCannotCompleteRising_fb.sts.value, Message := 'Partial fresh delay cannot complete transition');
        BadQualityCannotCompleteRising_clock(IN := FALSE); BadQualityCannotCompleteRising_phase := 3;
    END_IF;
3:
    BadQualityCannotCompleteRising_clock(IN := TRUE, PT := T#150MS); BadQualityCannotCompleteRising_fb();
    IF BadQualityCannotCompleteRising_clock.Q THEN
        AssertEquals_BOOL(Expected := TRUE, Actual := BadQualityCannotCompleteRising_fb.sts.value, Message := 'Full fresh delay completes transition');
        BadQualityCannotCompleteRising_done := TRUE; TEST_FINISHED();
    END_IF;
END_CASE;
END_METHOD

METHOD BadQualityCannotCompleteFalling
IF BadQualityCannotCompleteFalling_done THEN RETURN; END_IF;
TEST('BadQualityCannotCompleteFalling');
CASE BadQualityCannotCompleteFalling_phase OF
0:
    BadQualityCannotCompleteFalling_fb(inSignal := TRUE);
    BadQualityCannotCompleteFalling_fb.cfg.debounceOn := T#80MS; BadQualityCannotCompleteFalling_fb.cfg.debounceOff := T#80MS;
    BadQualityCannotCompleteFalling_fb(inSignal := FALSE);
    BadQualityCannotCompleteFalling_fb(inpQuality := TcForge.E_IO_Quality.BAD);
    BadQualityCannotCompleteFalling_phase := 1;
1:
    BadQualityCannotCompleteFalling_clock(IN := TRUE, PT := T#150MS); BadQualityCannotCompleteFalling_fb();
    IF BadQualityCannotCompleteFalling_clock.Q THEN
        AssertEquals_BOOL(Expected := TRUE, Actual := BadQualityCannotCompleteFalling_fb.sts.value, Message := 'Invalid elapsed time must hold established state');
        AssertFalse(Condition := BadQualityCannotCompleteFalling_fb.sts.risingEdge OR BadQualityCannotCompleteFalling_fb.sts.fallingEdge, Message := 'Invalid sample cannot emit edges');
        BadQualityCannotCompleteFalling_clock(IN := FALSE); BadQualityCannotCompleteFalling_fb(inpQuality := TcForge.E_IO_Quality.GOOD);
        AssertEquals_BOOL(Expected := TRUE, Actual := BadQualityCannotCompleteFalling_fb.sts.value, Message := 'Recovery starts a full fresh transition delay');
        BadQualityCannotCompleteFalling_phase := 2;
    END_IF;
2:
    BadQualityCannotCompleteFalling_clock(IN := TRUE, PT := T#30MS); BadQualityCannotCompleteFalling_fb();
    IF BadQualityCannotCompleteFalling_clock.Q THEN
        AssertEquals_BOOL(Expected := TRUE, Actual := BadQualityCannotCompleteFalling_fb.sts.value, Message := 'Partial fresh delay cannot complete transition');
        BadQualityCannotCompleteFalling_clock(IN := FALSE); BadQualityCannotCompleteFalling_phase := 3;
    END_IF;
3:
    BadQualityCannotCompleteFalling_clock(IN := TRUE, PT := T#150MS); BadQualityCannotCompleteFalling_fb();
    IF BadQualityCannotCompleteFalling_clock.Q THEN
        AssertEquals_BOOL(Expected := FALSE, Actual := BadQualityCannotCompleteFalling_fb.sts.value, Message := 'Full fresh delay completes transition');
        BadQualityCannotCompleteFalling_done := TRUE; TEST_FINISHED();
    END_IF;
END_CASE;
END_METHOD

METHOD ConfigChangeDiscardsDebounceCredit
IF ConfigChangeDiscardsDebounceCredit_done THEN RETURN; END_IF;
TEST('ConfigChangeDiscardsDebounceCredit');
CASE ConfigChangeDiscardsDebounceCredit_phase OF
0:
    ConfigChangeDiscardsDebounceCredit_fb.cfg.debounceOn := T#100MS;
    ConfigChangeDiscardsDebounceCredit_fb(inSignal := TRUE);
    ConfigChangeDiscardsDebounceCredit_phase := 1;
1:
    ConfigChangeDiscardsDebounceCredit_clock(IN := TRUE, PT := T#60MS); ConfigChangeDiscardsDebounceCredit_fb();
    IF ConfigChangeDiscardsDebounceCredit_clock.Q THEN
        ConfigChangeDiscardsDebounceCredit_fb.cfg.debounceOn := T#80MS;
        ConfigChangeDiscardsDebounceCredit_fb(); ConfigChangeDiscardsDebounceCredit_clock(IN := FALSE);
        ConfigChangeDiscardsDebounceCredit_phase := 2;
    END_IF;
2:
    ConfigChangeDiscardsDebounceCredit_clock(IN := TRUE, PT := T#30MS); ConfigChangeDiscardsDebounceCredit_fb();
    IF ConfigChangeDiscardsDebounceCredit_clock.Q THEN
        AssertFalse(Condition := ConfigChangeDiscardsDebounceCredit_fb.sts.value, Message := 'New delay cannot inherit old timer credit');
        ConfigChangeDiscardsDebounceCredit_done := TRUE; TEST_FINISHED();
    END_IF;
END_CASE;
END_METHOD

METHOD ReassignmentAndInvalidConfigHold
VAR fb : TcForge.FB_DigitalInput; END_VAR

TEST('ReassignmentAndInvalidConfigHold');
fb(inSignal := TRUE); AssertTrue(Condition := fb.sts.value, Message := 'Fixture has established TRUE');
fb(inpQuality := TcForge.E_IO_Quality.UNKNOWN); fb.cfg.invert := TRUE; fb();
AssertTrue(Condition := fb.sts.value, Message := 'Inversion cannot reinterpret invalid held raw');
AssertFalse(Condition := fb.sts.risingEdge OR fb.sts.fallingEdge, Message := 'Config edit under bad quality has no edge');
fb.ReassignInput();
AssertEquals_INT(Expected := 0, Actual := fb.sts.quality, Message := 'Reassignment immediately invalidates old source');
AssertFalse(Condition := fb.sts.value OR fb.sts.rawValue OR fb.sts.risingEdge OR fb.sts.fallingEdge, Message := 'Reassignment clears old history without an edge');
fb(); AssertEquals_INT(Expected := 0, Actual := fb.sts.quality, Message := 'Unknown adapter quality remains unknown');
fb(inpQuality := TcForge.E_IO_Quality.GOOD, inSignal := FALSE);
AssertTrue(Condition := fb.sts.value AND fb.sts.risingEdge, Message := 'Fresh source is conditioned using current inversion');
TEST_FINISHED();
END_METHOD

END_FUNCTION_BLOCK

// ---- Testing/Tests/FB_AlarmValidity_Test.TcPOU
FUNCTION_BLOCK FB_AlarmValidity_Test EXTENDS TcUnit.FB_TestSuite
VAR
    done : BOOL;
    restoredUnacked : FB_AlarmRestart_Probe;
    restoredAcked : FB_AlarmRestart_Probe;
    criteriaThreshold : TcForge.FB_AlarmThreshold;
    criteriaDeviation : TcForge.FB_AlarmDeviation;
    criteriaPhase : UINT;
    beforeChange : TON;
    afterChange : TON;
    reassignedRate : TcForge.FB_AlarmRateOfChange;
    severityAlarm : TcForge.FB_AlarmSimple;
    signalingAlarm : TcForge.FB_AlarmThreshold;
    recovery : TcForge.FB_AlarmSimple;
    phase : UINT;
    waitTimer : TON;
    clearTimer : TON;
    device0 : TcForge.FB_AlarmThreshold;
    device1 : TcForge.FB_AlarmThreshold;
    device2 : TcForge.FB_AlarmSimple;
    device3 : TcForge.FB_AlarmSimple;
    device4 : TcForge.FB_AlarmDeviation;
    device5 : TcForge.FB_AlarmDeviation;
    device6 : TcForge.FB_AlarmRateOfChange;
    device7 : TcForge.FB_AlarmRateOfChange;
    device8 : TcForge.FB_AlarmRateOfChange;
    device9 : TcForge.FB_AlarmLimit;
END_VAR

IF NOT done THEN
InvalidInputPreservesAlarm();
RestoredLatchPublishesSeverity();
RestoredAcknowledgmentNeedsClearEvidence();
InvalidConfigPreservesLatch();
RequireAckChangePreservesLatch();
SimpleValidityGate();
DeviationExtremeArithmetic();
DeviationRejectsBadBounds();
RateExtremeArithmetic();
RateRecoveryNeedsTwoSamples();
RateConfigReseedsHistory();
LimitRollupValidity();
InvalidSeverityPreservesAlarm();
SignalingNaNIsClassified();
RateReassignmentDropsHistory();
done := TRUE;
END_IF;
RecoveryHonorsFreshClearDelay();
CriteriaChangeRestartsTripDelay();

METHOD PRIVATE RestoredLatchPublishesSeverity
TEST('RestoredLatchPublishesSeverity');
restoredUnacked.SeedSavedLatch(acknowledged := FALSE);
restoredUnacked.cfg.common.bEnable := TRUE;
restoredUnacked.cfg.common.bRequireAck := TRUE;
restoredUnacked.cfg.common.eSeverity := TcForge.E_AlarmSeverity.SHUTDOWN;
restoredUnacked(inpActive := FALSE, inpValid := FALSE);
AssertTrue(restoredUnacked.sts.active AND restoredUnacked.sts.latched, 'Restored unacked latch remains active without valid input');
AssertFalse(restoredUnacked.sts.valid, 'Restored latch is not valid process evidence');
AssertEquals_DINT(TcForge.E_AlarmSeverity.SHUTDOWN, restoredUnacked.sts.eSeverity, 'Startup publishes configured severity despite invalid input');
restoredUnacked.cfg.common.eSeverity := TcForge.E_AlarmSeverity.INFO;
restoredUnacked();
AssertEquals_DINT(TcForge.E_AlarmSeverity.SHUTDOWN, restoredUnacked.sts.eSeverity, 'Later invalid evaluation preserves established severity');
restoredUnacked(inpValid := TRUE);
AssertTrue(restoredUnacked.sts.active AND restoredUnacked.sts.latched, 'Valid clear evidence alone cannot erase an unacked restored latch');
restoredUnacked.Ack(); restoredUnacked();
AssertFalse(restoredUnacked.sts.active, 'Explicit Ack and valid clear release restored latch');
TEST_FINISHED();
END_METHOD

METHOD PRIVATE RestoredAcknowledgmentNeedsClearEvidence
TEST('RestoredAcknowledgmentNeedsClearEvidence');
restoredAcked.SeedSavedLatch(acknowledged := TRUE);
restoredAcked.cfg.common.bEnable := TRUE;
restoredAcked.cfg.common.bRequireAck := TRUE;
restoredAcked.cfg.common.eSeverity := TcForge.E_AlarmSeverity.CRITICAL;
restoredAcked(inpActive := FALSE, inpValid := FALSE);
AssertTrue(restoredAcked.sts.active AND restoredAcked.sts.acked, 'Restored acknowledgment cannot clear alarm with invalid evidence');
AssertFalse(restoredAcked.sts.latched, 'Restored acknowledged alarm does not demand another Ack');
AssertEquals_DINT(TcForge.E_AlarmSeverity.CRITICAL, restoredAcked.sts.eSeverity, 'Acknowledged restored alarm retains meaningful startup severity');
restoredAcked(inpValid := TRUE);
AssertFalse(restoredAcked.sts.active OR restoredAcked.sts.acked, 'Valid clear evidence releases restored acknowledged latch without a second Ack');
TEST_FINISHED();
END_METHOD

METHOD PRIVATE InvalidInputPreservesAlarm
VAR bits : TcForge.U_IoRaw_Out; tripped, cleared : LTIME; END_VAR
TEST('InvalidInputPreservesAlarm');
device0.cfg.common.bEnable := TRUE; device0.cfg.bFailHigh := TRUE;
device0.cfg.common.eSeverity := TcForge.E_AlarmSeverity.CRITICAL;
device0(inpValue := 10.0); tripped := device0.sts.tsTripped; cleared := device0.sts.tsCleared;
bits.dw := DWORD#16#7FC00000; device0(inpValue := bits.fReal);
AssertTrue(device0.sts.active, 'NaN cannot clear active alarm');
AssertFalse(device0.sts.valid, 'NaN evaluation is invalid');
AssertEquals_DINT(TcForge.E_AlarmEvaluation.InvalidInput, device0.sts.evaluationState, 'NaN classified without FPU operation');
AssertEquals_DINT(TcForge.E_AlarmSeverity.CRITICAL, device0.sts.eSeverity, 'Established severity preserved');
AssertTrue(device0.sts.tsTripped = tripped AND device0.sts.tsCleared = cleared, 'Invalid evaluation creates no alarm edges');
TEST_FINISHED();
END_METHOD

METHOD PRIVATE InvalidConfigPreservesLatch
VAR bits : TcForge.U_IoRaw_Out; tripped, cleared : LTIME; END_VAR
TEST('InvalidConfigPreservesLatch');
device1.cfg.common.bEnable := TRUE; device1.cfg.bFailHigh := TRUE; device1.cfg.common.bRequireAck := TRUE;
device1(inpValue := 10.0);
bits.dw := DWORD#16#7FC00000; device1.cfg.fThreshold := bits.fReal;
device1(); device1.Ack(); device1();
AssertTrue(device1.sts.active, 'Ack during invalid config cannot clear latch');
AssertTrue(device1.sts.acked, 'Ack is recorded while evaluation is invalid');
device1.cfg.fThreshold := 20.0; device1();
AssertFalse(device1.sts.active, 'Valid clear evidence releases acknowledged latch');
TEST_FINISHED();
END_METHOD

METHOD PRIVATE RequireAckChangePreservesLatch
VAR bits : TcForge.U_IoRaw_Out; tripped, cleared : LTIME; END_VAR
TEST('RequireAckChangePreservesLatch');
device2.cfg.common.bEnable := TRUE; device2.cfg.common.bRequireAck := TRUE;
device2(inpActive := TRUE); device2.cfg.common.bRequireAck := FALSE; device2(inpActive := FALSE);
AssertTrue(device2.sts.active AND device2.sts.latched, 'Changing future latch policy does not erase unacked trip');
device2.Ack(); device2(); AssertFalse(device2.sts.active, 'Ack and valid clear release old latch');
TEST_FINISHED();
END_METHOD

METHOD PRIVATE SimpleValidityGate
VAR bits : TcForge.U_IoRaw_Out; tripped, cleared : LTIME; END_VAR
TEST('SimpleValidityGate');
device3.cfg.common.bEnable := TRUE; device3(inpActive := TRUE);
device3(inpActive := FALSE, inpValid := FALSE);
AssertTrue(device3.sts.active, 'Missing digital quality holds established alarm');
AssertFalse(device3.sts.valid, 'Missing quality is visible');
device3(inpValid := TRUE); AssertFalse(device3.sts.active, 'Valid clear evidence releases nonlatched alarm');
TEST_FINISHED();
END_METHOD

METHOD PRIVATE DeviationExtremeArithmetic
VAR bits : TcForge.U_IoRaw_Out; tripped, cleared : LTIME; END_VAR
TEST('DeviationExtremeArithmetic');
device4.cfg.common.bEnable := TRUE; device4.cfg.bUseSetpoint := TRUE;
device4.cfg.fHighLimit := 3.0E38; device4.cfg.fLowLimit := 3.0E38;
device4(inpPv := 3.0E38, inpSetpoint := 3.0E38);
AssertTrue(device4.sts.valid, 'Finite extremes use wide intermediate bounds');
AssertFalse(device4.sts.active, 'Large valid setpoint window contains PV');
TEST_FINISHED();
END_METHOD

METHOD PRIVATE DeviationRejectsBadBounds
VAR bits : TcForge.U_IoRaw_Out; tripped, cleared : LTIME; END_VAR
TEST('DeviationRejectsBadBounds');
device5.cfg.common.bEnable := TRUE; device5.cfg.fHighLimit := 1.0; device5.cfg.fLowLimit := 2.0; device5();
AssertEquals_DINT(TcForge.E_AlarmEvaluation.InvalidConfig, device5.sts.evaluationState, 'Reversed absolute bounds rejected');
device5.cfg.bUseSetpoint := TRUE; device5.cfg.fLowLimit := -1.0; device5();
AssertFalse(device5.sts.valid, 'Negative setpoint deviation rejected');
device5.cfg.fLowLimit := 1.0; bits.dw := DWORD#16#7F800000; device5(inpSetpoint := bits.fReal);
AssertEquals_DINT(TcForge.E_AlarmEvaluation.InvalidInput, device5.sts.evaluationState, 'Infinite active setpoint rejected');
TEST_FINISHED();
END_METHOD

METHOD PRIVATE RateExtremeArithmetic
VAR bits : TcForge.U_IoRaw_Out; tripped, cleared : LTIME; END_VAR
TEST('RateExtremeArithmetic');
device6.cfg.common.bEnable := TRUE; device6.cfg.fRateLimit := 1.0;
device6(inpPv := -3.0E38);
AssertEquals_DINT(TcForge.E_AlarmEvaluation.Initializing, device6.sts.evaluationState, 'First valid sample is baseline only');
device6(inpPv := 3.0E38);
AssertTrue(device6.sts.valid AND device6.sts.active, 'Extreme REAL step is valid LREAL rate');
AssertTrue(TcForge.F_IsFiniteLReal(device6.outRateOfChange), 'Rate remains finite');
AssertTrue(device6.outRateOfChange > LREAL#3.4E38, 'Rate is not narrowed or silently saturated');
TEST_FINISHED();
END_METHOD

METHOD PRIVATE RateRecoveryNeedsTwoSamples
VAR bits : TcForge.U_IoRaw_Out; tripped, cleared : LTIME; END_VAR
TEST('RateRecoveryNeedsTwoSamples');
device7.cfg.common.bEnable := TRUE; device7.cfg.fRateLimit := 1.0;
device7(inpPv := 0.0); device7(inpPv := 10.0);
AssertTrue(device7.sts.active, 'Rate trip established');
bits.dw := DWORD#16#7FC00000; device7(inpPv := bits.fReal);
AssertTrue(device7.sts.active, 'Invalid sample preserves rate alarm');
device7(inpPv := 10.0);
AssertEquals_DINT(TcForge.E_AlarmEvaluation.Initializing, device7.sts.evaluationState, 'Recovery reseeds history');
AssertTrue(device7.sts.active, 'Seed sample cannot clear prior trip');
device7(inpPv := 10.0);
AssertTrue(device7.sts.valid, 'Second valid sample supplies rate');
AssertFalse(device7.sts.active, 'Valid zero rate clears nonlatched trip');
TEST_FINISHED();
END_METHOD

METHOD PRIVATE RateConfigReseedsHistory
VAR bits : TcForge.U_IoRaw_Out; tripped, cleared : LTIME; END_VAR
TEST('RateConfigReseedsHistory');
device8.cfg.common.bEnable := TRUE; device8(inpPv := 0.0); device8(inpPv := 1.0);
device8.cfg.fRateLimit := -1.0; device8();
AssertEquals_DINT(TcForge.E_AlarmEvaluation.InvalidConfig, device8.sts.evaluationState, 'Negative rate limit rejected');
device8.cfg.fRateLimit := 2.0; device8(inpPv := 1000.0);
AssertEquals_DINT(TcForge.E_AlarmEvaluation.Initializing, device8.sts.evaluationState, 'Valid config recovery resets old sample');
device8(inpPv := 1000.0); AssertFalse(device8.sts.active, 'No synthetic rate across invalid configuration');
TEST_FINISHED();
END_METHOD

METHOD PRIVATE LimitRollupValidity
VAR bits : TcForge.U_IoRaw_Out; tripped, cleared : LTIME; END_VAR
TEST('LimitRollupValidity');
device9.cfg.Hi.common.bEnable := TRUE; device9.cfg.Hi.bFailHigh := TRUE;
device9(inpPv := 10.0); AssertTrue(device9.sts.valid, 'Disabled unused levels do not invalidate enabled tier');
device9(inpValid := FALSE);
AssertFalse(device9.sts.valid, 'Composite propagates invalid signal');
AssertTrue(device9.sts.anyActive, 'Composite preserves established tier alarm');
AssertEquals_DINT(TcForge.E_AlarmEvaluation.InvalidInput, device9.sts.Hi.evaluationState, 'Child exposes invalid signal');
device9.cfg.Hi.common.bEnable := FALSE; device9();
AssertEquals_DINT(TcForge.E_AlarmEvaluation.Disabled, device9.sts.evaluationState, 'All disabled is distinct from valid');
TEST_FINISHED();
END_METHOD

METHOD PRIVATE RecoveryHonorsFreshClearDelay
IF phase = 4 THEN RETURN; END_IF;
TEST('RecoveryHonorsFreshClearDelay');
CASE phase OF
0:
    recovery.cfg.common.bEnable := TRUE;
    recovery.cfg.common.tOffDelay := T#60MS;
    recovery(inpActive := TRUE);
    AssertTrue(recovery.sts.active, 'Trip established before quality loss');
    phase := 1;
1:
    recovery(inpActive := FALSE, inpValid := FALSE);
    waitTimer(IN := TRUE, PT := T#100MS);
    AssertTrue(recovery.sts.active, 'Invalid interval cannot count as clear evidence');
    IF waitTimer.Q THEN phase := 2; END_IF;
2:
    recovery(inpValid := TRUE);
    AssertTrue(recovery.sts.active, 'First valid clear sample starts full off-delay');
    clearTimer(IN := TRUE, PT := T#90MS);
    phase := 3;
3:
    recovery(); clearTimer(IN := TRUE, PT := T#90MS);
    IF clearTimer.ET < T#40MS THEN AssertTrue(recovery.sts.active, 'Recovery cannot release before fresh delay'); END_IF;
    IF clearTimer.Q THEN
        AssertFalse(recovery.sts.active, 'Sustained valid clear releases after off-delay');
        phase := 4; TEST_FINISHED();
    END_IF;
END_CASE;
END_METHOD

METHOD PRIVATE InvalidSeverityPreservesAlarm
VAR badSeverity : USINT := 255; END_VAR
TEST('InvalidSeverityPreservesAlarm');
severityAlarm.cfg.common.bEnable := TRUE;
severityAlarm.cfg.common.eSeverity := TcForge.E_AlarmSeverity.WARNING;
severityAlarm(inpActive := TRUE);
MEMCPY(ADR(severityAlarm.cfg.common.eSeverity), ADR(badSeverity), SIZEOF(badSeverity));
severityAlarm(inpActive := FALSE);
AssertEquals_DINT(TcForge.E_AlarmEvaluation.InvalidConfig, severityAlarm.sts.evaluationState, 'Unknown severity is invalid config');
AssertTrue(severityAlarm.sts.active, 'Invalid severity cannot clear established trip');
AssertEquals_DINT(TcForge.E_AlarmSeverity.WARNING, severityAlarm.sts.eSeverity, 'Established severity preserved');
TEST_FINISHED();
END_METHOD

METHOD PRIVATE SignalingNaNIsClassified
VAR bits : TcForge.U_IoRaw_Out; END_VAR
TEST('SignalingNaNIsClassified');
signalingAlarm.cfg.common.bEnable := TRUE; signalingAlarm.cfg.bFailHigh := TRUE;
bits.dw := DWORD#16#7F800001;
signalingAlarm(inpValue := bits.fReal);
AssertEquals_DINT(TcForge.E_AlarmEvaluation.InvalidInput, signalingAlarm.sts.evaluationState, 'Signaling NaN rejected before floating operations');
TEST_FINISHED();
END_METHOD

METHOD PRIVATE RateReassignmentDropsHistory
TEST('RateReassignmentDropsHistory');
reassignedRate.cfg.common.bEnable := TRUE; reassignedRate.cfg.fRateLimit := 1.0;
reassignedRate(inpPv := 0.0); reassignedRate(inpPv := 10.0);
AssertTrue(reassignedRate.sts.active, 'Rate alarm initially active');
reassignedRate.ReassignInput();
AssertFalse(reassignedRate.sts.valid, 'Reassignment invalidates immediately');
AssertTrue(reassignedRate.sts.active, 'Reassignment cannot clear established alarm');
reassignedRate(inpPv := 1000.0);
AssertEquals_DINT(TcForge.E_AlarmEvaluation.Initializing, reassignedRate.sts.evaluationState, 'New source starts with baseline sample');
reassignedRate(inpPv := 1000.0);
AssertFalse(reassignedRate.sts.active, 'Second fresh source sample supplies valid zero rate');
TEST_FINISHED();
END_METHOD

METHOD PRIVATE CriteriaChangeRestartsTripDelay
IF criteriaPhase = 4 THEN RETURN; END_IF;
TEST('CriteriaChangeRestartsTripDelay');
CASE criteriaPhase OF
0:
    criteriaThreshold.cfg.common.bEnable := TRUE;
    criteriaThreshold.cfg.common.tOnDelay := T#120MS;
    criteriaThreshold.cfg.bFailHigh := TRUE;
    criteriaDeviation.cfg.common.bEnable := TRUE;
    criteriaDeviation.cfg.common.tOnDelay := T#120MS;
    criteriaDeviation.cfg.fHighLimit := 1.0;
    criteriaPhase := 1;
1:
    criteriaThreshold(inpValue := 10.0); criteriaDeviation(inpPv := 10.0);
    beforeChange(IN := TRUE, PT := T#80MS);
    IF beforeChange.Q THEN
        criteriaThreshold.cfg.fThreshold := 1.0;
        criteriaDeviation.cfg.fHighLimit := 2.0;
        criteriaPhase := 2;
    END_IF;
2:
    criteriaThreshold(); criteriaDeviation();
    afterChange(IN := TRUE, PT := T#160MS);
    AssertFalse(criteriaThreshold.sts.active, 'New threshold cannot inherit old on-delay credit');
    AssertFalse(criteriaDeviation.sts.active, 'New deviation bounds cannot inherit old on-delay credit');
    IF afterChange.ET >= T#60MS THEN criteriaPhase := 3; END_IF;
3:
    criteriaThreshold(); criteriaDeviation();
    afterChange(IN := TRUE, PT := T#160MS);
    IF afterChange.Q THEN
        AssertTrue(criteriaThreshold.sts.active, 'New threshold trips after fresh full delay');
        AssertTrue(criteriaDeviation.sts.active, 'New deviation trips after fresh full delay');
        criteriaPhase := 4; TEST_FINISHED();
    END_IF;
END_CASE;
END_METHOD

END_FUNCTION_BLOCK

// ---- Testing/POUs/FB_AlarmRestart_Probe.TcPOU
// Injects restored flags into an otherwise fresh instance. This exercises
// startup policy, not actual TwinCAT persistent-image durability.
FUNCTION_BLOCK FB_AlarmRestart_Probe EXTENDS TcForge.FB_AlarmSimple

SUPER^();

METHOD PUBLIC SeedSavedLatch
VAR_INPUT acknowledged : BOOL; END_VAR
_latchedSync := TRUE;
_ackedSync := acknowledged;
END_METHOD

END_FUNCTION_BLOCK

// ---- Testing/Tests/FB_FilterLifecycle_Test.TcPOU
FUNCTION_BLOCK FB_FilterLifecycle_Test EXTENDS TcUnit.FB_TestSuite
VAR _done : BOOL; END_VAR

IF _done THEN RETURN; END_IF;
ScalingChangeReseedsInCurrentUnits();
TauOnlyChangeRetainsHistory();
ReenabledFilterReseedsFreshSample();
RawBypassReturnReseedsScaledSample();
PendingReseedWaitsForUsableSample();
SourceReassignmentInvalidatesHeldIdentity();
RawTypeChangeReseedsFreshInterpretation();
ExplicitSeedRejectsExceptionalBits();
_done := TRUE;

METHOD ScalingChangeReseedsInCurrentUnits
VAR fb : TcForge.FB_AnalogInput; held : REAL; END_VAR
TEST('ScalingChangeReseedsInCurrentUnits');
fb.cfg.inputType := __SYSTEM.TYPE_CLASS.TYPE_REAL;
fb.cfg.rawMax := 100.0;
fb.cfg.filterTau := T#1S;
fb.inRaw.fReal := 80.0;
fb();
held := fb.sts.value;
AssertTrue(Condition := held > 0.0 AND held < 80.0, Message := 'Initial configured filtering remains zero seeded');
fb.cfg.euMax := 1000.0;
fb();
AssertTrue(Condition := ABS(fb.sts.value - 800.0) < 0.001, Message := 'Scale change cannot blend old engineering units');
fb.inRaw.fReal := 0.0; fb();
AssertTrue(Condition := fb.sts.value > 0.0 AND fb.sts.value < 800.0, Message := 'Subsequent samples filter normally after reseed');
TEST_FINISHED();
END_METHOD

METHOD TauOnlyChangeRetainsHistory
VAR fb : TcForge.FB_AnalogInput; held : REAL; END_VAR
TEST('TauOnlyChangeRetainsHistory');
fb.cfg.inputType := __SYSTEM.TYPE_CLASS.TYPE_REAL;
fb.cfg.rawMax := 100.0;
fb.cfg.filterTau := T#1S;
fb.inRaw.fReal := 80.0;
fb();
held := fb.sts.value;
fb.cfg.filterTau := T#2S; fb();
AssertTrue(Condition := fb.sts.value > held AND fb.sts.value < 80.0, Message := 'Tau tuning changes response without reseeding');
TEST_FINISHED();
END_METHOD

METHOD ReenabledFilterReseedsFreshSample
VAR fb : TcForge.FB_AnalogInput; held : REAL; END_VAR
TEST('ReenabledFilterReseedsFreshSample');
fb.cfg.inputType := __SYSTEM.TYPE_CLASS.TYPE_REAL;
fb.cfg.rawMax := 100.0;
fb.cfg.filterTau := T#1S;
fb.inRaw.fReal := 80.0;
fb();
held := fb.sts.value;
fb.cfg.filterTau := T#0MS; fb.inRaw.fReal := 40.0; fb();
AssertTrue(Condition := fb.sts.value = 40.0, Message := 'Disabled filtering passes fresh scaled value');
fb.cfg.filterTau := T#1S; fb.inRaw.fReal := 60.0; fb();
AssertTrue(Condition := fb.sts.value = 60.0, Message := 'Reenabled filtering cannot reuse old history');
TEST_FINISHED();
END_METHOD

METHOD RawBypassReturnReseedsScaledSample
VAR fb : TcForge.FB_AnalogInput; held : REAL; END_VAR
TEST('RawBypassReturnReseedsScaledSample');
fb.cfg.inputType := __SYSTEM.TYPE_CLASS.TYPE_REAL;
fb.cfg.rawMax := 100.0;
fb.cfg.filterTau := T#1S;
fb.inRaw.fReal := 80.0;
fb();
held := fb.sts.value;
fb.cfg.useRawValue := TRUE; fb.inRaw.fReal := 45.0; fb();
AssertTrue(Condition := fb.sts.value = 45.0, Message := 'Bypass uses fresh raw value');
fb.cfg.useRawValue := FALSE; fb.inRaw.fReal := 30.0; fb();
AssertTrue(Condition := fb.sts.value = 30.0, Message := 'Leaving bypass seeds current scaled input');
TEST_FINISHED();
END_METHOD

METHOD PendingReseedWaitsForUsableSample
VAR fb : TcForge.FB_AnalogInput; held : REAL; END_VAR
TEST('PendingReseedWaitsForUsableSample');
fb.cfg.inputType := __SYSTEM.TYPE_CLASS.TYPE_REAL;
fb.cfg.rawMax := 100.0;
fb.cfg.filterTau := T#1S;
fb.inRaw.fReal := 80.0;
fb();
held := fb.sts.value;
fb.cfg.euMax := 200.0; fb.inRaw.fReal := 30.0;
fb(inpQuality := TcForge.E_IO_Quality.BAD); fb();
AssertTrue(Condition := fb.sts.value = held, Message := 'Bad quality preserves last output while configuration changes');
fb.cfg.rawMax := 0.0; fb(inpQuality := TcForge.E_IO_Quality.GOOD);
AssertTrue(Condition := fb.sts.value = held AND fb.IsFaulted(), Message := 'Invalid scaling cannot consume pending reseed');
fb.cfg.rawMax := 100.0; fb();
AssertTrue(Condition := fb.sts.value = 60.0 AND NOT fb.IsFaulted(), Message := 'First usable sample after repair performs pending reseed');
TEST_FINISHED();
END_METHOD

METHOD SourceReassignmentInvalidatesHeldIdentity
VAR fb : TcForge.FB_AnalogInput; held : REAL; END_VAR
TEST('SourceReassignmentInvalidatesHeldIdentity');
fb.cfg.inputType := __SYSTEM.TYPE_CLASS.TYPE_REAL;
fb.cfg.rawMax := 100.0;
fb.cfg.filterTau := T#1S;
fb.inRaw.fReal := 80.0;
fb();
held := fb.sts.value;
fb.ReassignInput();
AssertEquals_DINT(Expected := TcForge.E_IO_Quality.UNKNOWN, Actual := fb.sts.quality, Message := 'Reassignment immediately invalidates previous source quality');
AssertTrue(Condition := fb.sts.value = 0.0 AND fb.sts.rawReal = 0.0 AND fb.sts.scaled = 0.0, Message := 'Previous source measurements are no longer published');
fb(inpQuality := TcForge.E_IO_Quality.UNKNOWN);
AssertTrue(Condition := fb.sts.value = 0.0, Message := 'Waiting for source cannot restore previous measurement');
fb.inRaw.fReal := 25.0; fb(inpQuality := TcForge.E_IO_Quality.GOOD);
AssertTrue(Condition := fb.sts.value = 25.0, Message := 'Same-config new source gets fresh history');
fb.inRaw.fReal := 0.0; fb();
AssertTrue(Condition := fb.sts.value > 0.0 AND fb.sts.value < 25.0, Message := 'New source then follows normal filtering');
TEST_FINISHED();
END_METHOD

METHOD RawTypeChangeReseedsFreshInterpretation
VAR fb : TcForge.FB_AnalogInput; held : REAL; END_VAR
TEST('RawTypeChangeReseedsFreshInterpretation');
fb.cfg.inputType := __SYSTEM.TYPE_CLASS.TYPE_REAL;
fb.cfg.rawMax := 100.0;
fb.cfg.filterTau := T#1S;
fb.inRaw.fReal := 80.0;
fb();
held := fb.sts.value;
fb.cfg.inputType := __SYSTEM.TYPE_CLASS.TYPE_INT;
fb.inRaw.nInt := 20; fb();
AssertTrue(Condition := fb.sts.value = 20.0, Message := 'Raw representation change cannot reuse prior history');
TEST_FINISHED();
END_METHOD

METHOD ExplicitSeedRejectsExceptionalBits
VAR filter : TcForge.FB_LPF_FirstOrder_IIR; invalidBits : ULINT; invalid : LREAL; END_VAR
TEST('ExplicitSeedRejectsExceptionalBits');
filter.Seed(value := 30.0);
invalidBits := ULINT#16#7FF8000000000000;
Tc2_System.MEMCPY(destAddr := ADR(invalid), srcAddr := ADR(invalidBits), n := SIZEOF(invalid));
AssertFalse(Condition := filter.Seed(value := invalid), Message := 'NaN seed rejected without floating exception');
AssertTrue(Condition := filter.fOutput = 30.0, Message := 'Rejected seed leaves output unchanged');
filter(fInput := 10.0, fDt := 1.0, fTau := 1.0);
AssertTrue(Condition := filter.fOutput = 20.0, Message := 'Rejected seed also preserves history');
TEST_FINISHED();
END_METHOD

END_FUNCTION_BLOCK

// ---- Testing/Tests/FB_PolicyNumeric_Test.TcPOU
FUNCTION_BLOCK FB_PolicyNumeric_Test EXTENDS TcUnit.FB_TestSuite
VAR _done : BOOL; END_VAR

IF _done THEN RETURN; END_IF;
PermissiveRevokesExistingBypass();
PermissionRestoreDoesNotRestoreBypass();
InterlockRevocationPreservesLatchedFailure();
InterlockResetPreservesAuthorizedBypass();
FilterRejectsNaNAndRecovers();
FilterRejectsNonfiniteTiming();
FilterRejectsInfinityDuringBypass();
FilterHandlesOppositeFiniteExtremes();
FilterHandlesLargeFiniteTiming();
RealFiniteClassificationHandlesExceptionalBits();
LRealFiniteClassificationHandlesExceptionalBits();
_done := TRUE;

METHOD PermissiveRevokesExistingBypass
VAR fb : TcForge.FB_Permissives; END_VAR
TEST('PermissiveRevokesExistingBypass');
fb.cfg.nRequired := 1; fb.cfg.nBypassable := 1;
fb.MapInput(bitIndex := 0, inputValue := FALSE); fb();
fb.SetBypass(bitIndex := 0, bEnable := TRUE); fb();
AssertTrue(Condition := fb.sts.bOK, Message := 'Precondition: authorized bypass suppresses mapped false condition');
fb.cfg.nBypassable := 0; fb();
AssertFalse(Condition := fb.sts.bOK OR fb.sts.aFaceplates[0].bypassed, Message := 'Revocation immediately removes effective bypass');
AssertTrue(Condition := fb.sts.nBypassMask = 0, Message := 'Revoked bypass intent is erased');
TEST_FINISHED();
END_METHOD

METHOD PermissionRestoreDoesNotRestoreBypass
VAR fb : TcForge.FB_Permissives; END_VAR
TEST('PermissionRestoreDoesNotRestoreBypass');
fb.cfg.nBypassable := 1; fb.MapInput(bitIndex := 0, inputValue := FALSE);
fb.SetBypass(bitIndex := 0, bEnable := TRUE); fb();
fb.cfg.nBypassable := 0; fb();
fb.cfg.nBypassable := 1; fb();
AssertFalse(Condition := fb.sts.bOK, Message := 'Reauthorizing permission does not silently re-enable bypass');
fb.SetBypass(bitIndex := 0, bEnable := TRUE); fb();
AssertTrue(Condition := fb.sts.bOK, Message := 'Explicit new bypass remains available');
TEST_FINISHED();
END_METHOD

METHOD InterlockRevocationPreservesLatchedFailure
VAR fb : TcForge.FB_Interlock; END_VAR
TEST('InterlockRevocationPreservesLatchedFailure');
fb.cfg.nRequired := 1; fb.cfg.nBypassable := 1;
fb.MapInput(bitIndex := 0, inputValue := FALSE); fb();
fb.SetBypass(bitIndex := 0, bEnable := TRUE); fb();
AssertTrue(Condition := fb.sts.bOK, Message := 'Precondition: authorized interlock bypass');
fb.cfg.nBypassable := 0; fb();
AssertFalse(Condition := fb.sts.bOK, Message := 'Revocation exposes latched bad condition immediately');
fb.MapInput(bitIndex := 0, inputValue := TRUE); fb();
fb.cfg.nBypassable := 1; fb();
AssertFalse(Condition := fb.sts.bOK, Message := 'Healthy signal and renewed permission do not release latch');
fb.Reset(); fb.MapInput(bitIndex := 0, inputValue := TRUE); fb();
AssertTrue(Condition := fb.sts.bOK AND fb.sts.nBypassMask = 0, Message := 'Healthy explicit Reset recovers without resurrecting bypass');
TEST_FINISHED();
END_METHOD

METHOD InterlockResetPreservesAuthorizedBypass
VAR fb : TcForge.FB_Interlock; END_VAR
TEST('InterlockResetPreservesAuthorizedBypass');
fb.cfg.nBypassable := 1; fb.MapInput(bitIndex := 0, inputValue := FALSE);
fb.SetBypass(bitIndex := 0, bEnable := TRUE); fb(); fb.Reset(); fb();
AssertTrue(Condition := fb.sts.bOK AND fb.sts.nBypassMask = 1, Message := 'Reset deliberately preserves still-authorized bypass');
TEST_FINISHED();
END_METHOD

METHOD FilterRejectsNaNAndRecovers
VAR fb : TcForge.FB_LPF_FirstOrder_IIR; invalid : LREAL; invalidBits : ULINT; END_VAR
TEST('FilterRejectsNaNAndRecovers');
fb(fInput := 10.0, fDt := 1.0, fTau := 1.0);
invalidBits := ULINT#16#7FF8000000000000;
Tc2_System.MEMCPY(destAddr := ADR(invalid), srcAddr := ADR(invalidBits), n := SIZEOF(invalid));
fb(fInput := invalid, fDt := 1.0, fTau := 1.0);
AssertTrue(Condition := fb.bError AND fb.fOutput = 5.0, Message := 'NaN sample holds finite history and reports error');
fb(fInput := 10.0, fDt := 1.0, fTau := 1.0);
AssertTrue(Condition := NOT fb.bError AND ABS(fb.fOutput - 7.5) < 1E-9, Message := 'Valid sample recovers without poisoned history');
TEST_FINISHED();
END_METHOD

METHOD FilterRejectsNonfiniteTiming
VAR fb : TcForge.FB_LPF_FirstOrder_IIR; invalid : LREAL; invalidBits : ULINT; END_VAR
TEST('FilterRejectsNonfiniteTiming');
fb(fInput := 10.0, fDt := 1.0, fTau := 1.0);
invalidBits := ULINT#16#7FF8000000000000;
Tc2_System.MEMCPY(destAddr := ADR(invalid), srcAddr := ADR(invalidBits), n := SIZEOF(invalid));
fb(fInput := 50.0, fDt := invalid, fTau := 1.0);
AssertTrue(Condition := fb.bError AND fb.fOutput = 5.0, Message := 'NaN timing cannot poison state');
invalidBits := ULINT#16#7FF0000000000000;
Tc2_System.MEMCPY(destAddr := ADR(invalid), srcAddr := ADR(invalidBits), n := SIZEOF(invalid));
fb(fInput := 50.0, fDt := 1.0, fTau := invalid);
AssertTrue(Condition := fb.bError AND fb.fOutput = 5.0, Message := 'Infinite timing is rejected explicitly');
TEST_FINISHED();
END_METHOD

METHOD FilterRejectsInfinityDuringBypass
VAR fb : TcForge.FB_LPF_FirstOrder_IIR; invalid : LREAL; invalidBits : ULINT; END_VAR
TEST('FilterRejectsInfinityDuringBypass');
fb(fInput := 8.0, fDt := 0.0, fTau := 1.0);
invalidBits := ULINT#16#7FF0000000000000;
Tc2_System.MEMCPY(destAddr := ADR(invalid), srcAddr := ADR(invalidBits), n := SIZEOF(invalid));
fb(fInput := invalid, fDt := 0.0, fTau := 1.0);
AssertTrue(Condition := fb.bError AND fb.fOutput = 8.0, Message := 'Pass-through cannot copy nonfinite input into history');
TEST_FINISHED();
END_METHOD

METHOD FilterHandlesOppositeFiniteExtremes
VAR fb : TcForge.FB_LPF_FirstOrder_IIR; END_VAR
TEST('FilterHandlesOppositeFiniteExtremes');
fb(fInput := LREAL#1.7E308, fDt := 0.0, fTau := 1.0);
fb(fInput := LREAL#-1.7E308, fDt := 1.0, fTau := 1.0);
AssertTrue(Condition := NOT fb.bError AND ABS(fb.fOutput) < LREAL#1E292, Message := 'Finite opposite extremes average without subtraction overflow');
TEST_FINISHED();
END_METHOD

METHOD FilterHandlesLargeFiniteTiming
VAR fb : TcForge.FB_LPF_FirstOrder_IIR; END_VAR
TEST('FilterHandlesLargeFiniteTiming');
fb(fInput := 10.0, fDt := LREAL#1.7E308, fTau := LREAL#1.7E308);
AssertTrue(Condition := NOT fb.bError AND ABS(fb.fOutput - 5.0) < 1E-9, Message := 'Large finite timing preserves ratio without sum overflow');
TEST_FINISHED();
END_METHOD

METHOD RealFiniteClassificationHandlesExceptionalBits
VAR sample : REAL; bits : DWORD; END_VAR
TEST('RealFiniteClassificationHandlesExceptionalBits');
bits := DWORD#16#7F800000;
Tc2_System.MEMCPY(destAddr := ADR(sample), srcAddr := ADR(bits), n := SIZEOF(sample));
AssertFalse(Condition := TcForge.F_IsFiniteReal(value := sample), Message := 'Reject exponent-all-ones without floating arithmetic');
bits := DWORD#16#FF800000;
Tc2_System.MEMCPY(destAddr := ADR(sample), srcAddr := ADR(bits), n := SIZEOF(sample));
AssertFalse(Condition := TcForge.F_IsFiniteReal(value := sample), Message := 'Reject exponent-all-ones without floating arithmetic');
bits := DWORD#16#7FC00000;
Tc2_System.MEMCPY(destAddr := ADR(sample), srcAddr := ADR(bits), n := SIZEOF(sample));
AssertFalse(Condition := TcForge.F_IsFiniteReal(value := sample), Message := 'Reject exponent-all-ones without floating arithmetic');
bits := DWORD#16#7F800001;
Tc2_System.MEMCPY(destAddr := ADR(sample), srcAddr := ADR(bits), n := SIZEOF(sample));
AssertFalse(Condition := TcForge.F_IsFiniteReal(value := sample), Message := 'Reject exponent-all-ones without floating arithmetic');
bits := 1;
Tc2_System.MEMCPY(destAddr := ADR(sample), srcAddr := ADR(bits), n := SIZEOF(sample));
AssertTrue(Condition := TcForge.F_IsFiniteReal(value := sample), Message := 'Subnormal is finite');
AssertTrue(Condition := TcForge.F_IsFiniteReal(value := 0.0), Message := 'Zero is finite');
TEST_FINISHED();
END_METHOD

METHOD LRealFiniteClassificationHandlesExceptionalBits
VAR sample : LREAL; bits : ULINT; END_VAR
TEST('LRealFiniteClassificationHandlesExceptionalBits');
bits := ULINT#16#7FF0000000000000;
Tc2_System.MEMCPY(destAddr := ADR(sample), srcAddr := ADR(bits), n := SIZEOF(sample));
AssertFalse(Condition := TcForge.F_IsFiniteLReal(value := sample), Message := 'Reject exponent-all-ones without floating arithmetic');
bits := ULINT#16#FFF0000000000000;
Tc2_System.MEMCPY(destAddr := ADR(sample), srcAddr := ADR(bits), n := SIZEOF(sample));
AssertFalse(Condition := TcForge.F_IsFiniteLReal(value := sample), Message := 'Reject exponent-all-ones without floating arithmetic');
bits := ULINT#16#7FF8000000000000;
Tc2_System.MEMCPY(destAddr := ADR(sample), srcAddr := ADR(bits), n := SIZEOF(sample));
AssertFalse(Condition := TcForge.F_IsFiniteLReal(value := sample), Message := 'Reject exponent-all-ones without floating arithmetic');
bits := ULINT#16#7FF0000000000001;
Tc2_System.MEMCPY(destAddr := ADR(sample), srcAddr := ADR(bits), n := SIZEOF(sample));
AssertFalse(Condition := TcForge.F_IsFiniteLReal(value := sample), Message := 'Reject exponent-all-ones without floating arithmetic');
bits := 1;
Tc2_System.MEMCPY(destAddr := ADR(sample), srcAddr := ADR(bits), n := SIZEOF(sample));
AssertTrue(Condition := TcForge.F_IsFiniteLReal(value := sample), Message := 'Subnormal is finite');
AssertTrue(Condition := TcForge.F_IsFiniteLReal(value := 0.0), Message := 'Zero is finite');
TEST_FINISHED();
END_METHOD

END_FUNCTION_BLOCK

// ---- Testing/Tests/FB_OutputConfiguration_Test.TcPOU
FUNCTION_BLOCK FB_OutputConfiguration_Test EXTENDS TcUnit.FB_TestSuite
VAR
    done : BOOL;
    trustDigitalBackupImageRejected : FB_OutputRestart_Probe;
    trustDigitalMissingImageRejected : FB_OutputRestart_Probe;
    trustDigitalFreshCommandWithUntrustedImage : FB_OutputRestart_Probe;
    trustAnalogBackupImageRejected : FB_AnalogOutputRestart_Probe;
    trustAnalogMissingImageRejected : FB_AnalogOutputRestart_Probe;
    trustAnalogFreshCommandWithUntrustedImage : FB_AnalogOutputRestart_Probe;

    restartDigitalNoSavedIntent : FB_OutputRestart_Probe;
    restartDigitalValidZeroIntent : FB_OutputRestart_Probe;
    restartDigitalResetDiscardsSavedIntent : FB_OutputRestart_Probe;
    restartDigitalForceSafeDiscardsSavedIntent : FB_OutputRestart_Probe;
    restartDigitalConfigDiscardsSavedIntent : FB_OutputRestart_Probe;
    restartAnalogNoSavedIntent : FB_AnalogOutputRestart_Probe;
    restartAnalogValidZeroIntent : FB_AnalogOutputRestart_Probe;
    restartAnalogResetDiscardsSavedIntent : FB_AnalogOutputRestart_Probe;
    restartAnalogForceSafeDiscardsSavedIntent : FB_AnalogOutputRestart_Probe;
    restartAnalogConfigDiscardsSavedIntent : FB_AnalogOutputRestart_Probe;

    nanConfigOutput : TcForge.FB_AnalogOutput;
    nanFallbackOutput : TcForge.FB_AnalogOutput;
    nanCommandOutput : TcForge.FB_AnalogOutput;
    infiniteOutput : TcForge.FB_AnalogOutput;
    delayedMailbox : TcForge.FB_OperatorMailbox;
    urgentMailbox : TcForge.FB_OperatorMailbox;
    device0 : TcForge.FB_DigitalOutput;
    device1 : TcForge.FB_DigitalOutput;
    device2 : TcForge.FB_DigitalOutput;
    device3 : TcForge.FB_DigitalOutput;
    device4 : TcForge.FB_DigitalOutput;
    device5 : TcForge.FB_DigitalOutput;
    device6 : TcForge.FB_AnalogOutput;
    device7 : TcForge.FB_AnalogOutput;
    device8 : TcForge.FB_AnalogOutput;
    device9 : TcForge.FB_AnalogOutput;
    device10 : TcForge.FB_AnalogOutput;
    device11 : TcForge.FB_TwoPosActuator;
    device12 : TcForge.FB_TwoPosActuator;
    device13 : TcForge.FB_TwoPosActuator;
    device14 : TcForge.FB_TwoPosActuator;
    device15 : TcForge.FB_TwoPosActuator;
END_VAR

IF done THEN RETURN; END_IF;
DigitalInvertDiscardsOff();
DigitalTimingDiscardsPulse();
DigitalFreshCommandBeforeScan();
DigitalFallbackOverridesQualityHold();
DigitalQueuedOffCancelled();
DigitalSafeLevelIsElectrical();
AnalogScalingDiscardsCommand();
AnalogFreshTypeCommand();
AnalogQueuedValueCancelled();
AnalogUnitMetadataPreservesIntent();
AnalogConfigRecoveryKeepsFault();
ActuatorHoldChangeRequiresCommand();
ActuatorTimeoutChangeStopsTravel();
ActuatorFreshCommandBeforeScan();
ActuatorQueuedTravelCancelled();
ActuatorConfigRecoveryKeepsFault();
DelayedSetOffCancellation();
UrgentCommandsSurviveConfigurationBarrier();
AnalogNaNConfigurationAndRecovery();
AnalogNaNSafeRawUsesZero();
AnalogNaNCommandsRejected();
AnalogInfinityRejected();
DigitalNoSavedIntent();
DigitalValidZeroIntent();
DigitalResetDiscardsSavedIntent();
DigitalForceSafeDiscardsSavedIntent();
DigitalConfigDiscardsSavedIntent();
AnalogNoSavedIntent();
AnalogValidZeroIntent();
AnalogResetDiscardsSavedIntent();
AnalogForceSafeDiscardsSavedIntent();
AnalogConfigDiscardsSavedIntent();
DigitalBackupImageRejected();
DigitalMissingImageRejected();
DigitalFreshCommandWithUntrustedImage();
AnalogBackupImageRejected();
AnalogMissingImageRejected();
AnalogFreshCommandWithUntrustedImage();
done := TRUE;

METHOD PRIVATE DigitalInvertDiscardsOff
VAR rsp : TcForge.E_RpcMethodResponse; END_VAR
TEST('DigitalInvertDiscardsOff');
device0.SetOff(); device0();
device0.cfg.invert := TRUE; device0();
AssertFalse(device0.outSignal, 'Inversion change cannot reinterpret previous SetOff');
AssertTrue(device0.sts.outputInhibited, 'Changed output remains inhibited');
device0.SetOff(); device0();
AssertTrue(device0.outSignal, 'Fresh SetOff explicitly commands inverted electrical high');
TEST_FINISHED();
END_METHOD

METHOD PRIVATE DigitalTimingDiscardsPulse
VAR rsp : TcForge.E_RpcMethodResponse; END_VAR
TEST('DigitalTimingDiscardsPulse');
device1.cfg.mode := TcForge.E_DigitalOutput_Mode.SinglePulse;
device1.cfg.pulseOn := T#10S;
device1.SetOn(); device1();
AssertTrue(device1.outSignal, 'Initial pulse is active');
device1.cfg.pulseOn := T#20S; device1();
AssertFalse(device1.outSignal, 'Changed timing discards pulse intent');
device1.SetOn(); device1();
AssertTrue(device1.outSignal, 'Fresh command creates a fresh pulse edge');
TEST_FINISHED();
END_METHOD

METHOD PRIVATE DigitalFreshCommandBeforeScan
VAR rsp : TcForge.E_RpcMethodResponse; END_VAR
TEST('DigitalFreshCommandBeforeScan');
device2(); device2.cfg.invert := TRUE;
rsp := device2.SetOff(); device2();
AssertEquals_DINT(TcForge.E_RpcMethodResponse.ACCEPTED, rsp, 'New-config command accepted before cycle');
AssertTrue(device2.outSignal, 'Cycle preserves newly accepted command');
TEST_FINISHED();
END_METHOD

METHOD PRIVATE DigitalFallbackOverridesQualityHold
VAR rsp : TcForge.E_RpcMethodResponse; END_VAR
TEST('DigitalFallbackOverridesQualityHold');
device3.cfg.holdOnBadQuality := TRUE;
device3.SetOn(); device3(); device3(inpQuality := TcForge.E_IO_Quality.BAD);
AssertTrue(device3.outSignal, 'Explicit quality hold retains previous terminal level');
device3.cfg.debounceOn := T#1S; device3();
AssertFalse(device3.outSignal, 'Configuration invalidation overrides quality hold');
TEST_FINISHED();
END_METHOD

METHOD PRIVATE DigitalQueuedOffCancelled
VAR rsp : TcForge.E_RpcMethodResponse; END_VAR
TEST('DigitalQueuedOffCancelled');
device4();
rsp := device4.OperatorSetOff(requestId := 901);
AssertEquals_DINT(TcForge.E_RpcMethodResponse.QUEUED, rsp, 'Off queued under old config');
device4.cfg.invert := TRUE; device4();
rsp := device4.OperatorCommandResult(requestId := 901);
AssertEquals_DINT(TcForge.E_RpcMethodResponse.CANCELLED, rsp, 'Old inverted-off interpretation is cancelled');
AssertFalse(device4.outSignal, 'Queued off cannot energize after inversion changes');
TEST_FINISHED();
END_METHOD

METHOD PRIVATE DigitalSafeLevelIsElectrical
VAR rsp : TcForge.E_RpcMethodResponse; END_VAR
TEST('DigitalSafeLevelIsElectrical');
device5.SetOn(); device5(); device5.cfg.safeOutput := TRUE; device5();
AssertTrue(device5.outSignal, 'Explicit safe electrical level applies');
AssertTrue(device5.sts.outputInhibited, 'Electrical high fallback is still inhibited operating intent');
TEST_FINISHED();
END_METHOD

METHOD PRIVATE AnalogScalingDiscardsCommand
VAR rsp : TcForge.E_RpcMethodResponse; END_VAR
TEST('AnalogScalingDiscardsCommand');
device6.cfg.rawMax := 1000.0;
device6.SetValue(rValue := 50.0); device6();
AssertEquals_REAL(500.0, device6.sts.rawReal, 0.01, 'Initial scaling');
device6.cfg.rawMax := 2000.0; device6();
AssertEquals_REAL(0.0, device6.sts.rawReal, 0.01, 'Changed scale uses fallback');
AssertTrue(device6.sts.outputInhibited, 'Scaling change disarms');
device6.SetValue(rValue := 50.0); device6();
AssertEquals_REAL(1000.0, device6.sts.rawReal, 0.01, 'Fresh command uses new scaling');
TEST_FINISHED();
END_METHOD

METHOD PRIVATE AnalogFreshTypeCommand
VAR rsp : TcForge.E_RpcMethodResponse; END_VAR
TEST('AnalogFreshTypeCommand');
device7.SetValue(rValue := 50.0); device7();
device7.cfg.outputType := __SYSTEM.TYPE_CLASS.TYPE_REAL;
device7.cfg.useRawValue := TRUE;
device7.SetValue(rValue := 12.5); device7();
AssertEquals_REAL(12.5, device7.outRaw.fReal, 0.001, 'Fresh pre-cycle command uses new type');
AssertFalse(device7.sts.outputInhibited, 'New intent remains armed');
TEST_FINISHED();
END_METHOD

METHOD PRIVATE AnalogQueuedValueCancelled
VAR rsp : TcForge.E_RpcMethodResponse; END_VAR
TEST('AnalogQueuedValueCancelled');
device8(); device8.OperatorSetValue(requestId := 902, rValue := 50.0);
device8.cfg.useRawValue := TRUE; device8();
rsp := device8.OperatorCommandResult(requestId := 902);
AssertEquals_DINT(TcForge.E_RpcMethodResponse.CANCELLED, rsp, 'Queued old-scale value cancelled');
AssertTrue(device8.sts.outputInhibited, 'Cancelled queue cannot arm output');
TEST_FINISHED();
END_METHOD

METHOD PRIVATE AnalogUnitMetadataPreservesIntent
VAR rsp : TcForge.E_RpcMethodResponse; END_VAR
TEST('AnalogUnitMetadataPreservesIntent');
device9.cfg.useRawValue := TRUE; device9.SetValue(rValue := 25.0); device9();
AssertTrue(device9.sts.unit = TcForge.E_Unit.UNSPECIFIED, 'Default output unit is not guessed');
device9.cfg.unit := TcForge.E_Unit.DEGREE_CELSIUS; device9();
AssertTrue(device9.sts.unit = TcForge.E_Unit.DEGREE_CELSIUS, 'Status echoes configured unit');
AssertEquals_REAL(25.0, device9.sts.rawReal, 0.01, 'Display unit metadata does not alter electrical intent');
TEST_FINISHED();
END_METHOD

METHOD PRIVATE AnalogConfigRecoveryKeepsFault
VAR rsp : TcForge.E_RpcMethodResponse; END_VAR
TEST('AnalogConfigRecoveryKeepsFault');
device10.cfg.euMax := 0.0; device10();
AssertTrue(device10.IsFaulted(), 'Invalid config faults');
device10.cfg.euMax := 100.0; device10();
AssertTrue(device10.IsFaulted(), 'Correcting config does not acknowledge latched fault');
AssertTrue(device10.sts.outputInhibited, 'Fault recovery cannot restart output');
TEST_FINISHED();
END_METHOD

METHOD PRIVATE ActuatorHoldChangeRequiresCommand
VAR rsp : TcForge.E_RpcMethodResponse; END_VAR
TEST('ActuatorHoldChangeRequiresCommand');
device11(inAdvanced := TRUE); device11.Advance(); device11();
AssertFalse(device11.outAdvance, 'No hold after reaching advanced');
device11.cfg.holdAtAdvanced := TRUE; device11();
AssertFalse(device11.outAdvance, 'Enabling hold cannot revive completed travel intent');
rsp := device11.Advance(); device11();
AssertEquals_DINT(TcForge.E_RpcMethodResponse.ACCEPTED, rsp, 'Fresh command at inhibited position accepted');
AssertTrue(device11.outAdvance, 'Explicit new hold intent energizes advanced coil');
TEST_FINISHED();
END_METHOD

METHOD PRIVATE ActuatorTimeoutChangeStopsTravel
VAR rsp : TcForge.E_RpcMethodResponse; END_VAR
TEST('ActuatorTimeoutChangeStopsTravel');
device12(); device12.Advance(); device12();
AssertTrue(device12.outAdvance, 'Motion initially energized');
device12.cfg.advTimeoutS := 8; device12();
AssertFalse(device12.outAdvance, 'Timeout edits cancel active travel');
AssertFalse(device12.sts.moving, 'No stale travel state survives');
device12.Advance(); device12();
AssertTrue(device12.outAdvance, 'Fresh command starts travel again');
TEST_FINISHED();
END_METHOD

METHOD PRIVATE ActuatorFreshCommandBeforeScan
VAR rsp : TcForge.E_RpcMethodResponse; END_VAR
TEST('ActuatorFreshCommandBeforeScan');
device13(); device13.cfg.holdAtRetracted := TRUE;
rsp := device13.Retract(); device13(inRetracted := TRUE);
AssertEquals_DINT(TcForge.E_RpcMethodResponse.ACCEPTED, rsp, 'New-config retract accepted');
AssertTrue(device13.outRetract, 'New command remains valid through cycle');
TEST_FINISHED();
END_METHOD

METHOD PRIVATE ActuatorQueuedTravelCancelled
VAR rsp : TcForge.E_RpcMethodResponse; END_VAR
TEST('ActuatorQueuedTravelCancelled');
device14(); device14.OperatorAdvance(requestId := 903);
device14.cfg.advTimeoutS := 8; device14();
rsp := device14.OperatorCommandResult(requestId := 903);
AssertEquals_DINT(TcForge.E_RpcMethodResponse.CANCELLED, rsp, 'Old queued motion cancelled');
AssertFalse(device14.outAdvance, 'Cancelled command cannot move');
TEST_FINISHED();
END_METHOD

METHOD PRIVATE ActuatorConfigRecoveryKeepsFault
VAR rsp : TcForge.E_RpcMethodResponse; END_VAR
TEST('ActuatorConfigRecoveryKeepsFault');
device15(inAdvanced := TRUE, inRetracted := TRUE);
AssertTrue(device15.IsFaulted(), 'Contradictory feedback faults');
device15.cfg.holdAtAdvanced := TRUE; device15(inRetracted := FALSE);
AssertTrue(device15.IsFaulted(), 'Config change preserves latched feedback fault');
AssertFalse(device15.outAdvance, 'No hold while fault remains latched');
TEST_FINISHED();
END_METHOD

METHOD PRIVATE DelayedSetOffCancellation
VAR
    rsp : TcForge.E_RpcMethodResponse;
    consumed : BOOL;
    cmd : TcForge.E_OperatorCommand;
END_VAR
TEST('DelayedSetOffCancellation');
delayedMailbox.BeginConsume();
rsp := delayedMailbox.Submit(requestId := 910, command := TcForge.E_OperatorCommand.SetOff, value := 0.0);
AssertEquals_DINT(TcForge.E_RpcMethodResponse.QUEUED, rsp, 'Queue SetOff before configuration invalidation');
delayedMailbox.CancelNormal(includeSetOff := TRUE);
// Delaying reconciliation and another ordinary cancellation cannot erase the barrier.
delayedMailbox.CancelNormal();
rsp := delayedMailbox.Submit(requestId := 911, command := TcForge.E_OperatorCommand.SetOff, value := 0.0);
AssertEquals_DINT(TcForge.E_RpcMethodResponse.REJECTED_BUSY, rsp, 'New SetOff cannot cross unreconciled barrier');
consumed := delayedMailbox.BeginConsume(command => cmd);
AssertFalse(consumed, 'Old SetOff is cancelled before eventual consumption');
IF consumed THEN delayedMailbox.EndConsume(result := TcForge.E_RpcMethodResponse.ACCEPTED); END_IF;
rsp := delayedMailbox.GetResult(requestId := 910);
AssertEquals_DINT(TcForge.E_RpcMethodResponse.CANCELLED, rsp, 'Cancelled result retained');
rsp := delayedMailbox.Submit(requestId := 912, command := TcForge.E_OperatorCommand.SetOff, value := 0.0);
AssertEquals_DINT(TcForge.E_RpcMethodResponse.QUEUED, rsp, 'Fresh SetOff accepted after barrier reconciles');
consumed := delayedMailbox.BeginConsume(command => cmd);
AssertTrue(consumed, 'Fresh SetOff can execute');
IF consumed THEN delayedMailbox.EndConsume(result := TcForge.E_RpcMethodResponse.ACCEPTED); END_IF;
TEST_FINISHED();
END_METHOD

METHOD PRIVATE UrgentCommandsSurviveConfigurationBarrier
VAR
    rsp : TcForge.E_RpcMethodResponse;
    consumed : BOOL;
    cmd : TcForge.E_OperatorCommand;
END_VAR
TEST('UrgentCommandsSurviveConfigurationBarrier');
urgentMailbox.BeginConsume();
urgentMailbox.CancelNormal(includeSetOff := TRUE);
rsp := urgentMailbox.Submit(requestId := 913, command := TcForge.E_OperatorCommand.ForceSafe, value := 0.0);
AssertEquals_DINT(TcForge.E_RpcMethodResponse.QUEUED, rsp, 'ForceSafe crosses cancellation barrier');
consumed := urgentMailbox.BeginConsume(command => cmd);
AssertTrue(consumed, 'ForceSafe survives reconciliation');
AssertEquals_DINT(TcForge.E_OperatorCommand.ForceSafe, cmd, 'Correct urgent command');
IF consumed THEN urgentMailbox.EndConsume(result := TcForge.E_RpcMethodResponse.ACCEPTED); END_IF;
urgentMailbox.CancelNormal(includeSetOff := TRUE);
rsp := urgentMailbox.Submit(requestId := 914, command := TcForge.E_OperatorCommand.Abort, value := 0.0);
AssertEquals_DINT(TcForge.E_RpcMethodResponse.QUEUED, rsp, 'Abort crosses cancellation barrier');
consumed := urgentMailbox.BeginConsume(command => cmd);
AssertTrue(consumed, 'Abort survives reconciliation');
AssertEquals_DINT(TcForge.E_OperatorCommand.Abort, cmd, 'Correct abort command');
IF consumed THEN urgentMailbox.EndConsume(result := TcForge.E_RpcMethodResponse.ACCEPTED); END_IF;
TEST_FINISHED();
END_METHOD

METHOD PRIVATE AnalogNaNConfigurationAndRecovery
VAR
    bits : TcForge.U_IoRaw_Out;
    rsp : TcForge.E_RpcMethodResponse;
END_VAR
TEST('AnalogNaNConfigurationAndRecovery');
nanConfigOutput.SetValue(rValue := 50.0); nanConfigOutput();
bits.dw := DWORD#16#7FC00000;
nanConfigOutput.cfg.euMax := bits.fReal;
nanConfigOutput();
AssertTrue(nanConfigOutput.IsFaulted(), 'NaN scaling faults without FPU exception');
AssertEquals_REAL(0.0, nanConfigOutput.sts.rawReal, 0.001, 'NaN scaling uses finite fallback');
nanConfigOutput(); // Both current and prior snapshots contain NaN.
nanConfigOutput.cfg.euMax := 100.0;
nanConfigOutput(); // Previous snapshot contains NaN during recovery.
AssertTrue(nanConfigOutput.IsFaulted(), 'Finite recovery preserves configuration fault');
AssertTrue(nanConfigOutput.sts.outputInhibited, 'Finite recovery does not restart old intent');
TEST_FINISHED();
END_METHOD

METHOD PRIVATE AnalogNaNSafeRawUsesZero
VAR
    bits : TcForge.U_IoRaw_Out;
    rsp : TcForge.E_RpcMethodResponse;
END_VAR
TEST('AnalogNaNSafeRawUsesZero');
bits.dw := DWORD#16#7FC00000;
nanFallbackOutput.cfg.safeRaw := bits.fReal;
nanFallbackOutput(); nanFallbackOutput();
AssertTrue(nanFallbackOutput.IsFaulted(), 'NaN fallback is invalid configuration');
AssertEquals_DINT(0, nanFallbackOutput.outRaw.nInt, 'Unrepresentable fallback writes finite zero');
nanFallbackOutput.cfg.safeRaw := 12.0; nanFallbackOutput();
AssertEquals_DINT(12, nanFallbackOutput.outRaw.nInt, 'Corrected finite electrical fallback applies while faulted');
TEST_FINISHED();
END_METHOD

METHOD PRIVATE AnalogNaNCommandsRejected
VAR
    bits : TcForge.U_IoRaw_Out;
    rsp : TcForge.E_RpcMethodResponse;
END_VAR
TEST('AnalogNaNCommandsRejected');
nanCommandOutput.cfg.useRawValue := TRUE;
nanCommandOutput.SetValue(rValue := 12.0); nanCommandOutput();
bits.dw := DWORD#16#7FC00000;
rsp := nanCommandOutput.SetValue(rValue := bits.fReal);
AssertEquals_DINT(TcForge.E_RpcMethodResponse.REJECTED_INVALID_PARAMETER, rsp, 'Direct NaN rejected before float comparison');
rsp := nanCommandOutput.OperatorSetValue(requestId := 920, rValue := bits.fReal);
AssertEquals_DINT(TcForge.E_RpcMethodResponse.REJECTED_INVALID_PARAMETER, rsp, 'Mailbox NaN rejected before float comparison');
nanCommandOutput();
AssertEquals_REAL(12.0, nanCommandOutput.sts.rawReal, 0.001, 'Rejected NaN commands preserve valid prior intent');
TEST_FINISHED();
END_METHOD

METHOD PRIVATE AnalogInfinityRejected
VAR
    bits : TcForge.U_IoRaw_Out;
    rsp : TcForge.E_RpcMethodResponse;
END_VAR
TEST('AnalogInfinityRejected');
infiniteOutput();
bits.dw := DWORD#16#7F800000;
rsp := infiniteOutput.SetValue(rValue := bits.fReal);
AssertEquals_DINT(TcForge.E_RpcMethodResponse.REJECTED_INVALID_PARAMETER, rsp, 'Infinite command rejected');
infiniteOutput.cfg.rawMax := bits.fReal; infiniteOutput();
AssertTrue(infiniteOutput.IsFaulted(), 'Infinite scale faults before arithmetic');
AssertEquals_REAL(0.0, infiniteOutput.sts.rawReal, 0.001, 'Infinite scale writes finite fallback');
TEST_FINISHED();
END_METHOD

METHOD PRIVATE DigitalNoSavedIntent
TEST('DigitalNoSavedIntent');
restartDigitalNoSavedIntent.cfg.restoreCommandOnRestart := TRUE;
restartDigitalNoSavedIntent.cfg.invert := TRUE;
restartDigitalNoSavedIntent();
AssertTrue(restartDigitalNoSavedIntent.sts.outputInhibited, 'Missing or invalidated saved intent cannot arm after startup');
AssertFalse(restartDigitalNoSavedIntent.outSignal, 'Inversion cannot turn absent intent into electrical high');
TEST_FINISHED();
END_METHOD

METHOD PRIVATE DigitalValidZeroIntent
TEST('DigitalValidZeroIntent');
restartDigitalValidZeroIntent.cfg.restoreCommandOnRestart := TRUE;
restartDigitalValidZeroIntent.cfg.invert := TRUE;
restartDigitalValidZeroIntent.SetOff(); restartDigitalValidZeroIntent();
AssertFalse(restartDigitalValidZeroIntent.sts.outputInhibited, 'Accepted command initially arms output');
restartDigitalValidZeroIntent.SimulateStartup(); restartDigitalValidZeroIntent();
AssertFalse(restartDigitalValidZeroIntent.sts.outputInhibited, 'Saved zero command is valid intent');
AssertTrue(restartDigitalValidZeroIntent.outSignal, 'Accepted inverted SetOff restores electrical high');
TEST_FINISHED();
END_METHOD

METHOD PRIVATE DigitalResetDiscardsSavedIntent
TEST('DigitalResetDiscardsSavedIntent');
restartDigitalResetDiscardsSavedIntent.cfg.restoreCommandOnRestart := TRUE;
restartDigitalResetDiscardsSavedIntent.cfg.invert := TRUE;
restartDigitalResetDiscardsSavedIntent.SetOff(); restartDigitalResetDiscardsSavedIntent();
AssertFalse(restartDigitalResetDiscardsSavedIntent.sts.outputInhibited, 'Accepted command initially arms output');
restartDigitalResetDiscardsSavedIntent.Reset(); restartDigitalResetDiscardsSavedIntent();
restartDigitalResetDiscardsSavedIntent.SimulateStartup(); restartDigitalResetDiscardsSavedIntent();
AssertTrue(restartDigitalResetDiscardsSavedIntent.sts.outputInhibited, 'Missing or invalidated saved intent cannot arm after startup');
AssertFalse(restartDigitalResetDiscardsSavedIntent.outSignal, 'Inversion cannot turn absent intent into electrical high');
TEST_FINISHED();
END_METHOD

METHOD PRIVATE DigitalForceSafeDiscardsSavedIntent
TEST('DigitalForceSafeDiscardsSavedIntent');
restartDigitalForceSafeDiscardsSavedIntent.cfg.restoreCommandOnRestart := TRUE;
restartDigitalForceSafeDiscardsSavedIntent.cfg.invert := TRUE;
restartDigitalForceSafeDiscardsSavedIntent.SetOff(); restartDigitalForceSafeDiscardsSavedIntent();
AssertFalse(restartDigitalForceSafeDiscardsSavedIntent.sts.outputInhibited, 'Accepted command initially arms output');
restartDigitalForceSafeDiscardsSavedIntent.ForceSafe(); restartDigitalForceSafeDiscardsSavedIntent();
restartDigitalForceSafeDiscardsSavedIntent.SimulateStartup(); restartDigitalForceSafeDiscardsSavedIntent();
AssertTrue(restartDigitalForceSafeDiscardsSavedIntent.sts.outputInhibited, 'Missing or invalidated saved intent cannot arm after startup');
AssertFalse(restartDigitalForceSafeDiscardsSavedIntent.outSignal, 'Inversion cannot turn absent intent into electrical high');
TEST_FINISHED();
END_METHOD

METHOD PRIVATE DigitalConfigDiscardsSavedIntent
TEST('DigitalConfigDiscardsSavedIntent');
restartDigitalConfigDiscardsSavedIntent.cfg.restoreCommandOnRestart := TRUE;
restartDigitalConfigDiscardsSavedIntent.cfg.invert := TRUE;
restartDigitalConfigDiscardsSavedIntent.SetOff(); restartDigitalConfigDiscardsSavedIntent();
AssertFalse(restartDigitalConfigDiscardsSavedIntent.sts.outputInhibited, 'Accepted command initially arms output');
restartDigitalConfigDiscardsSavedIntent.cfg.qualityFaultAfter := T#2S; restartDigitalConfigDiscardsSavedIntent();
restartDigitalConfigDiscardsSavedIntent.SimulateStartup(); restartDigitalConfigDiscardsSavedIntent();
AssertTrue(restartDigitalConfigDiscardsSavedIntent.sts.outputInhibited, 'Missing or invalidated saved intent cannot arm after startup');
AssertFalse(restartDigitalConfigDiscardsSavedIntent.outSignal, 'Inversion cannot turn absent intent into electrical high');
TEST_FINISHED();
END_METHOD

METHOD PRIVATE AnalogNoSavedIntent
TEST('AnalogNoSavedIntent');
restartAnalogNoSavedIntent.cfg.restoreCommandOnRestart := TRUE;
restartAnalogNoSavedIntent.cfg.useRawValue := TRUE; restartAnalogNoSavedIntent.cfg.safeRaw := 17.0;
restartAnalogNoSavedIntent();
AssertTrue(restartAnalogNoSavedIntent.sts.outputInhibited, 'Missing or invalidated saved intent cannot arm after startup');
AssertEquals_REAL(17.0, restartAnalogNoSavedIntent.sts.rawReal, 0.001, 'Absent intent applies nonzero electrical fallback');
TEST_FINISHED();
END_METHOD

METHOD PRIVATE AnalogValidZeroIntent
TEST('AnalogValidZeroIntent');
restartAnalogValidZeroIntent.cfg.restoreCommandOnRestart := TRUE;
restartAnalogValidZeroIntent.cfg.useRawValue := TRUE; restartAnalogValidZeroIntent.cfg.safeRaw := 17.0;
restartAnalogValidZeroIntent.SetValue(rValue := 0.0); restartAnalogValidZeroIntent();
AssertFalse(restartAnalogValidZeroIntent.sts.outputInhibited, 'Accepted command initially arms output');
restartAnalogValidZeroIntent.SimulateStartup(); restartAnalogValidZeroIntent();
AssertFalse(restartAnalogValidZeroIntent.sts.outputInhibited, 'Saved zero command is valid intent');
AssertEquals_REAL(0.0, restartAnalogValidZeroIntent.sts.rawReal, 0.001, 'Accepted zero restores as a command');
TEST_FINISHED();
END_METHOD

METHOD PRIVATE AnalogResetDiscardsSavedIntent
TEST('AnalogResetDiscardsSavedIntent');
restartAnalogResetDiscardsSavedIntent.cfg.restoreCommandOnRestart := TRUE;
restartAnalogResetDiscardsSavedIntent.cfg.useRawValue := TRUE; restartAnalogResetDiscardsSavedIntent.cfg.safeRaw := 17.0;
restartAnalogResetDiscardsSavedIntent.SetValue(rValue := 0.0); restartAnalogResetDiscardsSavedIntent();
AssertFalse(restartAnalogResetDiscardsSavedIntent.sts.outputInhibited, 'Accepted command initially arms output');
restartAnalogResetDiscardsSavedIntent.Reset(); restartAnalogResetDiscardsSavedIntent();
restartAnalogResetDiscardsSavedIntent.SimulateStartup(); restartAnalogResetDiscardsSavedIntent();
AssertTrue(restartAnalogResetDiscardsSavedIntent.sts.outputInhibited, 'Missing or invalidated saved intent cannot arm after startup');
AssertEquals_REAL(17.0, restartAnalogResetDiscardsSavedIntent.sts.rawReal, 0.001, 'Absent intent applies nonzero electrical fallback');
TEST_FINISHED();
END_METHOD

METHOD PRIVATE AnalogForceSafeDiscardsSavedIntent
TEST('AnalogForceSafeDiscardsSavedIntent');
restartAnalogForceSafeDiscardsSavedIntent.cfg.restoreCommandOnRestart := TRUE;
restartAnalogForceSafeDiscardsSavedIntent.cfg.useRawValue := TRUE; restartAnalogForceSafeDiscardsSavedIntent.cfg.safeRaw := 17.0;
restartAnalogForceSafeDiscardsSavedIntent.SetValue(rValue := 0.0); restartAnalogForceSafeDiscardsSavedIntent();
AssertFalse(restartAnalogForceSafeDiscardsSavedIntent.sts.outputInhibited, 'Accepted command initially arms output');
restartAnalogForceSafeDiscardsSavedIntent.ForceSafe(); restartAnalogForceSafeDiscardsSavedIntent();
restartAnalogForceSafeDiscardsSavedIntent.SimulateStartup(); restartAnalogForceSafeDiscardsSavedIntent();
AssertTrue(restartAnalogForceSafeDiscardsSavedIntent.sts.outputInhibited, 'Missing or invalidated saved intent cannot arm after startup');
AssertEquals_REAL(17.0, restartAnalogForceSafeDiscardsSavedIntent.sts.rawReal, 0.001, 'Absent intent applies nonzero electrical fallback');
TEST_FINISHED();
END_METHOD

METHOD PRIVATE AnalogConfigDiscardsSavedIntent
TEST('AnalogConfigDiscardsSavedIntent');
restartAnalogConfigDiscardsSavedIntent.cfg.restoreCommandOnRestart := TRUE;
restartAnalogConfigDiscardsSavedIntent.cfg.useRawValue := TRUE; restartAnalogConfigDiscardsSavedIntent.cfg.safeRaw := 17.0;
restartAnalogConfigDiscardsSavedIntent.SetValue(rValue := 0.0); restartAnalogConfigDiscardsSavedIntent();
AssertFalse(restartAnalogConfigDiscardsSavedIntent.sts.outputInhibited, 'Accepted command initially arms output');
restartAnalogConfigDiscardsSavedIntent.cfg.qualityFaultAfter := T#2S; restartAnalogConfigDiscardsSavedIntent();
restartAnalogConfigDiscardsSavedIntent.SimulateStartup(); restartAnalogConfigDiscardsSavedIntent();
AssertTrue(restartAnalogConfigDiscardsSavedIntent.sts.outputInhibited, 'Missing or invalidated saved intent cannot arm after startup');
AssertEquals_REAL(17.0, restartAnalogConfigDiscardsSavedIntent.sts.rawReal, 0.001, 'Absent intent applies nonzero electrical fallback');
TEST_FINISHED();
END_METHOD

METHOD PRIVATE DigitalBackupImageRejected
TEST('DigitalBackupImageRejected');
trustDigitalBackupImageRejected.cfg.restoreCommandOnRestart := TRUE;
trustDigitalBackupImageRejected.cfg.invert := TRUE;
trustDigitalBackupImageRejected.SeedSavedCommand(value := FALSE);
trustDigitalBackupImageRejected.simulatedBootDataLoaded := TRUE;
trustDigitalBackupImageRejected.simulatedOldBootData := TRUE;
trustDigitalBackupImageRejected();
AssertTrue(trustDigitalBackupImageRejected.sts.outputInhibited, 'Untrusted persistent image cannot restore output');
AssertFalse(trustDigitalBackupImageRejected.outSignal, 'Electrical output honors startup trust');
trustDigitalBackupImageRejected.simulatedBootDataLoaded := TRUE; trustDigitalBackupImageRejected.simulatedOldBootData := FALSE;
trustDigitalBackupImageRejected.SimulateStartup(); trustDigitalBackupImageRejected();
AssertTrue(trustDigitalBackupImageRejected.sts.outputInhibited, 'Later trust cannot revive previously rejected saved intent');
TEST_FINISHED();
END_METHOD

